C05476=1184.490,135.905,-53.759,-178.491,6.283,148.692
C05477=1184.495,135.656,-53.738,-178.495,6.282,148.692
C05478=1184.501,135.407,-53.718,-178.497,6.280,148.693
C05479=1184.505,135.158,-53.698,-178.499,6.279,148.693
C05480=1184.509,134.909,-53.678,-178.502,6.277,148.694
C05481=1184.515,134.659,-53.657,-178.505,6.275,148.694
C05482=1184.519,134.410,-53.637,-178.508,6.274,148.695
C05483=1184.524,134.161,-53.617,-178.510,6.273,148.695
C05484=1184.529,133.912,-53.597,-178.513,6.271,148.695
C05485=1184.533,133.663,-53.577,-178.515,6.270,148.696
C05486=1184.538,133.414,-53.557,-178.519,6.268,148.696
C05487=1184.544,133.165,-53.536,-178.521,6.267,148.697
C05488=1184.548,132.897,-53.515,-178.523,6.266,148.697
C05489=1184.554,132.628,-53.493,-178.527,6.264,148.698
C05490=1184.559,132.359,-53.472,-178.529,6.262,148.698
C05491=1184.564,132.091,-53.449,-178.532,6.261,148.699
C05492=1184.569,131.841,-53.430,-178.535,6.259,148.699
C05493=1184.573,131.592,-53.409,-178.538,6.257,148.700
C05494=1184.578,131.342,-53.390,-178.540,6.257,148.700
C05495=1184.582,131.094,-53.369,-178.543,6.255,148.700
C05496=1184.587,130.844,-53.350,-178.546,6.253,148.701
C05497=1184.592,130.596,-53.330,-178.549,6.252,148.701
C05498=1184.597,130.346,-53.310,-178.551,6.251,148.702
C05499=1184.602,130.097,-53.289,-178.553,6.249,148.702
C05500=1184.607,129.847,-53.269,-178.557,6.248,148.703
C05501=1184.612,129.599,-53.249,-178.559,6.247,148.703
C05502=1184.617,129.349,-53.230,-178.561,6.245,148.704
C05503=1184.621,129.101,-53.209,-178.565,6.243,148.704
C05504=1184.626,128.851,-53.190,-178.567,6.242,148.705
C05505=1184.631,128.601,-53.170,-178.569,6.241,148.705
C05506=1184.636,128.353,-53.150,-178.572,6.239,148.705
C05507=1184.640,128.104,-53.130,-178.575,6.238,148.706
C05508=1184.645,127.855,-53.110,-178.577,6.237,148.706
C05509=1184.650,127.605,-53.090,-178.580,6.235,148.707
C05510=1184.655,127.356,-53.071,-178.583,6.233,148.707
C05511=1184.659,127.107,-53.051,-178.585,6.233,148.708
C05512=1184.664,126.858,-53.031,-178.588,6.231,148.708
C05513=1184.669,126.608,-53.011,-178.591,6.229,148.709
C05514=1184.674,126.360,-52.991,-178.593,6.227,148.709
C05515=1184.679,126.110,-52.972,-178.596,6.227,148.710
C05516=1184.683,125.861,-52.952,-178.599,6.225,148.710
C05517=1184.688,125.612,-52.932,-178.601,6.223,148.710
C05518=1184.693,125.363,-52.912,-178.604,6.223,148.711
C05519=1184.697,125.114,-52.893,-178.607,6.221,148.711
C05520=1184.702,124.865,-52.873,-178.609,6.219,148.712
C05521=1184.707,124.616,-52.854,-178.612,6.218,148.712
C05522=1184.712,124.366,-52.834,-178.615,6.217,148.713
C05523=1184.716,124.117,-52.814,-178.617,6.215,148.713
C05524=1184.721,123.867,-52.795,-178.620,6.214,148.714
C05525=1184.726,123.619,-52.775,-178.623,6.213,148.714
C05526=1184.731,123.369,-52.755,-178.625,6.211,148.715
C05527=1184.736,123.120,-52.735,-178.628,6.210,148.715
C05528=1184.741,122.871,-52.716,-178.630,6.208,148.716
C05529=1184.745,122.622,-52.697,-178.633,6.207,148.716
C05530=1184.749,122.373,-52.677,-178.636,6.206,148.717
C05531=1184.755,122.124,-52.657,-178.638,6.204,148.717
C05532=1184.760,121.874,-52.638,-178.641,6.203,148.718
C05533=1184.764,121.625,-52.618,-178.644,6.202,148.718
C05534=1184.770,121.376,-52.599,-178.646,6.200,148.718
C05535=1184.774,121.127,-52.580,-178.650,6.199,148.719
C05536=1184.779,120.878,-52.560,-178.652,6.198,148.719
C05537=1184.784,120.628,-52.541,-178.654,6.196,148.720
C05538=1184.788,120.379,-52.520,-178.657,6.194,148.720
C05539=1184.793,120.130,-52.501,-178.660,6.194,148.721
C05540=1184.797,119.881,-52.482,-178.662,6.192,148.721
C05541=1184.802,119.631,-52.462,-178.665,6.190,148.722
C05542=1184.808,119.383,-52.443,-178.668,6.190,148.722
C05543=1184.812,119.133,-52.423,-178.670,6.188,148.723
C05544=1184.818,118.884,-52.404,-178.673,6.186,148.723
C05545=1184.822,118.635,-52.385,-178.676,6.186,148.724
C05546=1184.826,118.385,-52.365,-178.678,6.184,148.724
C05547=1184.832,118.136,-52.346,-178.680,6.183,148.725
C05548=1184.837,117.887,-52.327,-178.684,6.182,148.725
C05549=1184.841,117.638,-52.308,-178.686,6.180,148.726
C05550=1184.846,117.389,-52.288,-178.689,6.179,148.726
C05551=1184.851,117.140,-52.269,-178.692,6.178,148.727
C05552=1184.855,116.891,-52.250,-178.694,6.176,148.727
C05553=1184.860,116.640,-52.231,-178.697,6.175,148.727
C05554=1184.866,116.392,-52.212,-178.700,6.174,148.728
C05555=1184.870,116.142,-52.192,-178.702,6.172,148.728
C05556=1184.875,115.893,-52.173,-178.705,6.171,148.729
C05557=1184.880,115.644,-52.154,-178.708,6.170,148.729
C05558=1184.885,115.395,-52.134,-178.710,6.169,148.730
C05559=1184.889,115.146,-52.115,-178.713,6.167,148.730
C05560=1184.894,114.897,-52.096,-178.716,6.165,148.731
C05561=1184.899,114.647,-52.076,-178.718,6.165,148.731
C05562=1184.904,114.398,-52.058,-178.721,6.163,148.732
C05563=1184.909,114.149,-52.039,-178.723,6.162,148.732
C05564=1184.913,113.900,-52.020,-178.726,6.161,148.733
C05565=1184.918,113.650,-52.000,-178.729,6.159,148.733
C05566=1184.923,113.402,-51.981,-178.731,6.158,148.734
C05567=1184.928,113.152,-51.963,-178.734,6.156,148.734
C05568=1184.933,112.903,-51.943,-178.736,6.156,148.735
C05569=1184.937,112.654,-51.924,-178.739,6.154,148.735
C05570=1184.942,112.405,-51.905,-178.742,6.152,148.736
C05571=1184.948,112.155,-51.886,-178.744,6.151,148.736
C05572=1184.952,111.906,-51.867,-178.747,6.150,148.737
C05573=1184.957,111.656,-51.848,-178.749,6.149,148.737
C05574=1184.961,111.408,-51.829,-178.753,6.148,148.738
C05575=1184.967,111.158,-51.810,-178.755,6.146,148.738
C05576=1184.971,110.909,-51.791,-178.757,6.145,148.739
C05577=1184.976,110.660,-51.772,-178.761,6.144,148.739
C05578=1184.982,110.410,-51.753,-178.763,6.143,148.740
C05579=1184.986,110.162,-51.734,-178.765,6.141,148.740
C05580=1184.991,109.912,-51.715,-178.769,6.140,148.741
C05581=1184.996,109.663,-51.697,-178.771,6.139,148.741
C05582=1185.001,109.413,-51.677,-178.773,6.137,148.741
C05583=1185.005,109.165,-51.658,-178.776,6.136,148.742
C05584=1185.010,108.914,-51.640,-178.779,6.135,148.743
C05585=1185.015,108.666,-51.621,-178.782,6.133,148.743
C05586=1185.020,108.417,-51.603,-178.784,6.132,148.744
C05587=1185.024,108.167,-51.583,-178.787,6.131,148.744
C05588=1185.029,107.919,-51.564,-178.789,6.130,148.745
C05589=1185.034,107.668,-51.546,-178.792,6.128,148.745
C05590=1185.039,107.420,-51.527,-178.794,6.127,148.745
C05591=1185.044,107.170,-51.508,-178.797,6.126,148.746
C05592=1185.049,106.902,-51.488,-178.800,6.124,148.746
C05593=1185.054,106.633,-51.468,-178.803,6.124,148.747
C05594=1185.060,106.366,-51.447,-178.806,6.122,148.748
C05595=1185.064,106.097,-51.427,-178.809,6.121,148.748
C05596=1185.070,105.847,-51.409,-178.812,6.119,148.749
C05597=1185.075,105.599,-51.390,-178.814,6.118,148.749
C05598=1185.079,105.349,-51.372,-178.817,6.117,148.750
C05599=1185.084,105.100,-51.352,-178.819,6.116,148.750
C05600=1185.089,104.850,-51.334,-178.822,6.114,148.751
C05601=1185.093,104.601,-51.315,-178.824,6.113,148.751
C05602=1185.099,104.352,-51.297,-178.827,6.112,148.752
C05603=1185.103,104.103,-51.278,-178.830,6.111,148.752
C05604=1185.108,103.853,-51.260,-178.833,6.110,148.753
C05605=1185.113,103.604,-51.241,-178.835,6.109,148.753
C05606=1185.117,103.355,-51.222,-178.838,6.107,148.754
C05607=1185.122,103.106,-51.204,-178.841,6.106,148.754
C05608=1185.128,102.857,-51.185,-178.843,6.105,148.755
C05609=1185.133,102.607,-51.167,-178.846,6.103,148.755
C05610=1185.137,102.358,-51.148,-178.848,6.103,148.756
C05611=1185.142,102.109,-51.129,-178.851,6.101,148.756
C05612=1185.147,101.860,-51.111,-178.854,6.100,148.757
C05613=1185.151,101.610,-51.093,-178.856,6.099,148.757
C05614=1185.157,101.361,-51.074,-178.859,6.098,148.758
C05615=1185.162,101.112,-51.056,-178.862,6.096,148.758
C05616=1185.166,100.862,-51.037,-178.864,6.096,148.759
C05617=1185.171,100.613,-51.019,-178.867,6.094,148.759
C05618=1185.176,100.364,-51.000,-178.869,6.093,148.760
C05619=1185.181,100.115,-50.982,-178.872,6.092,148.760
C05620=1185.185,99.865,-50.964,-178.874,6.091,148.761
C05621=1185.190,99.616,-50.945,-178.878,6.089,148.761
C05622=1185.196,99.367,-50.926,-178.880,6.088,148.762
C05623=1185.201,99.117,-50.908,-178.883,6.087,148.762
C05624=1185.205,98.868,-50.890,-178.886,6.085,148.763
C05625=1185.210,98.619,-50.871,-178.888,6.084,148.763
C05626=1185.214,98.370,-50.853,-178.891,6.083,148.764
C05627=1185.220,98.120,-50.835,-178.893,6.082,148.764
C05628=1185.224,97.870,-50.816,-178.896,6.081,148.765
C05629=1185.229,97.621,-50.798,-178.898,6.080,148.765
C05630=1185.234,97.372,-50.781,-178.902,6.078,148.766
C05631=1185.239,97.124,-50.762,-178.904,6.078,148.766
C05632=1185.244,96.874,-50.744,-178.906,6.076,148.767
C05633=1185.249,96.624,-50.725,-178.909,6.075,148.767
C05634=1185.254,96.375,-50.707,-178.912,6.074,148.768
C05635=1185.259,96.126,-50.689,-178.914,6.073,148.769
C05636=1185.264,95.877,-50.671,-178.917,6.071,148.769
C05637=1185.268,95.628,-50.653,-178.920,6.071,148.770
C05638=1185.273,95.378,-50.635,-178.922,6.069,148.770
C05639=1185.278,95.128,-50.617,-178.925,6.068,148.770
C05640=1185.283,94.879,-50.598,-178.928,6.067,148.771
C05641=1185.288,94.630,-50.579,-178.930,6.066,148.771
C05642=1185.293,94.381,-50.561,-178.933,6.065,148.772
C05643=1185.298,94.132,-50.543,-178.935,6.063,148.773
C05644=1185.302,93.882,-50.525,-178.938,6.063,148.773
C05645=1185.307,93.633,-50.507,-178.941,6.061,148.774
C05646=1185.312,93.384,-50.489,-178.943,6.061,148.774
C05647=1185.317,93.135,-50.471,-178.946,6.059,148.775
C05648=1185.322,92.885,-50.453,-178.949,6.058,148.775
C05649=1185.327,92.636,-50.435,-178.951,6.057,148.776
C05650=1185.332,92.387,-50.417,-178.953,6.056,148.776
C05651=1185.336,92.137,-50.399,-178.957,6.054,148.777
C05652=1185.341,91.887,-50.382,-178.959,6.053,148.777
C05653=1185.346,91.638,-50.364,-178.962,6.052,148.778
C05654=1185.351,91.389,-50.346,-178.964,6.051,148.778
C05655=1185.356,91.140,-50.328,-178.967,6.050,148.779
C05656=1185.361,90.891,-50.310,-178.969,6.049,148.779
C05657=1185.366,90.642,-50.292,-178.973,6.048,148.780
C05658=1185.371,90.392,-50.274,-178.975,6.047,148.780
C05659=1185.375,90.143,-50.255,-178.977,6.046,148.781
C05660=1185.380,89.893,-50.237,-178.980,6.044,148.781
C05661=1185.385,89.644,-50.219,-178.983,6.044,148.782
C05662=1185.390,89.394,-50.202,-178.985,6.042,148.783
C05663=1185.395,89.145,-50.184,-178.988,6.041,148.783
C05664=1185.400,88.896,-50.166,-178.991,6.040,148.784
C05665=1185.405,88.647,-50.148,-178.993,6.039,148.784
C05666=1185.410,88.398,-50.130,-178.996,6.038,148.785
C05667=1185.414,88.148,-50.112,-178.998,6.037,148.785
C05668=1185.420,87.899,-50.095,-179.001,6.035,148.786
C05669=1185.425,87.650,-50.077,-179.004,6.034,148.786
C05670=1185.430,87.400,-50.059,-179.006,6.034,148.787
C05671=1185.434,87.151,-50.042,-179.009,6.032,148.787
C05672=1185.439,86.902,-50.024,-179.012,6.032,148.788
C05673=1185.444,86.653,-50.006,-179.014,6.030,148.788
C05674=1185.449,86.403,-49.988,-179.017,6.029,148.789
C05675=1185.454,86.154,-49.970,-179.020,6.028,148.789
C05676=1185.459,85.904,-49.953,-179.022,6.027,148.790
C05677=1185.464,85.655,-49.935,-179.024,6.026,148.790
C05678=1185.469,85.406,-49.917,-179.028,6.025,148.791
C05679=1185.473,85.157,-49.901,-179.030,6.024,148.792
C05680=1185.478,84.907,-49.883,-179.033,6.022,148.792
C05681=1185.483,84.658,-49.865,-179.035,6.022,148.793
C05682=1185.488,84.408,-49.847,-179.038,6.020,148.793
C05683=1185.493,84.159,-49.829,-179.040,6.019,148.794
C05684=1185.498,83.910,-49.811,-179.043,6.019,148.794
C05685=1185.503,83.661,-49.795,-179.046,6.017,148.795
C05686=1185.507,83.411,-49.777,-179.048,6.016,148.795
C05687=1185.512,83.162,-49.759,-179.051,6.015,148.796
C05688=1185.518,82.912,-49.741,-179.054,6.014,148.796
C05689=1185.522,82.664,-49.724,-179.056,6.013,148.797
C05690=1185.527,82.414,-49.707,-179.059,6.012,148.798
C05691=1185.532,82.165,-49.689,-179.061,6.011,148.798
C05692=1185.537,81.915,-49.672,-179.064,6.010,148.799
C05693=1185.542,81.666,-49.654,-179.067,6.009,148.799
C05694=1185.546,81.417,-49.636,-179.070,6.007,148.800
C05695=1185.551,81.167,-49.619,-179.072,6.007,148.800
C05696=1185.556,80.899,-49.600,-179.075,6.005,148.801
C05697=1185.562,80.630,-49.581,-179.078,6.005,148.801
C05698=1185.567,80.362,-49.563,-179.080,6.003,148.802
C05699=1185.572,80.094,-49.544,-179.083,6.002,148.803
C05700=1185.577,79.844,-49.526,-179.086,6.001,148.803
C05701=1185.582,79.595,-49.508,-179.088,6.000,148.804
C05702=1185.587,79.345,-49.492,-179.091,6.000,148.804
C05703=1185.592,79.096,-49.474,-179.094,5.998,148.805
C05704=1185.597,78.846,-49.457,-179.096,5.997,148.805
C05705=1185.602,78.597,-49.440,-179.099,5.996,148.806
C05706=1185.607,78.348,-49.422,-179.102,5.995,148.806
C05707=1185.612,78.099,-49.405,-179.104,5.994,148.807
C05708=1185.616,77.850,-49.388,-179.107,5.993,148.807
C05709=1185.622,77.600,-49.370,-179.109,5.992,148.808
C05710=1185.627,77.350,-49.353,-179.112,5.991,148.809
C05711=1185.631,77.101,-49.336,-179.115,5.990,148.809
C05712=1185.636,76.851,-49.318,-179.117,5.989,148.810
C05713=1185.642,76.603,-49.301,-179.120,5.987,148.810
C05714=1185.646,76.353,-49.284,-179.123,5.987,148.811
C05715=1185.651,76.104,-49.267,-179.125,5.986,148.811
C05716=1185.656,75.855,-49.249,-179.128,5.985,148.812
C05717=1185.661,75.605,-49.232,-179.130,5.984,148.812
C05718=1185.666,75.355,-49.215,-179.133,5.983,148.813
C05719=1185.670,75.106,-49.198,-179.136,5.982,148.814
C05720=1185.676,74.857,-49.181,-179.138,5.981,148.814
C05721=1185.680,74.608,-49.164,-179.141,5.980,148.815
C05722=1185.686,74.358,-49.147,-179.143,5.979,148.815
C05723=1185.690,74.109,-49.129,-179.146,5.978,148.816
C05724=1185.695,73.859,-49.112,-179.149,5.976,148.816
C05725=1185.700,73.610,-49.095,-179.151,5.976,148.817
C05726=1185.705,73.361,-49.079,-179.153,5.975,148.817
C05727=1185.710,73.112,-49.061,-179.157,5.974,148.818
C05728=1185.715,72.862,-49.044,-179.159,5.973,148.818
C05729=1185.720,72.612,-49.027,-179.161,5.972,148.819
C05730=1185.725,72.363,-49.010,-179.164,5.970,148.819
C05731=1185.730,72.114,-48.992,-179.167,5.970,148.820
C05732=1185.734,71.865,-48.976,-179.169,5.969,148.821
C05733=1185.740,71.615,-48.958,-179.172,5.968,148.821
C05734=1185.744,71.366,-48.942,-179.175,5.967,148.822
C05735=1185.750,71.116,-48.925,-179.177,5.966,148.822
C05736=1185.754,70.867,-48.908,-179.180,5.965,148.823
C05737=1185.759,70.618,-48.891,-179.182,5.964,148.823
C05738=1185.764,70.368,-48.874,-179.185,5.963,148.824
C05739=1185.769,70.120,-48.857,-179.188,5.962,148.824
C05740=1185.774,69.870,-48.840,-179.190,5.961,148.825
C05741=1185.779,69.620,-48.823,-179.193,5.961,148.826
C05742=1185.784,69.370,-48.806,-179.196,5.959,148.826
C05743=1185.789,69.122,-48.790,-179.198,5.958,148.827
C05744=1185.794,68.872,-48.772,-179.200,5.958,148.827
C05745=1185.799,68.622,-48.756,-179.204,5.956,148.828
C05746=1185.803,68.373,-48.739,-179.206,5.955,148.828
C05747=1185.809,68.124,-48.722,-179.208,5.955,148.829
C05748=1185.813,67.874,-48.706,-179.211,5.953,148.829
C05749=1185.819,67.625,-48.688,-179.214,5.953,148.830
C05750=1185.824,67.376,-48.672,-179.216,5.952,148.831
C05751=1185.828,67.126,-48.655,-179.219,5.950,148.831
C05752=1185.833,66.876,-48.638,-179.222,5.950,148.832
C05753=1185.838,66.627,-48.621,-179.224,5.949,148.832
C05754=1185.843,66.378,-48.605,-179.227,5.948,148.833
C05755=1185.848,66.128,-48.588,-179.229,5.947,148.833
C05756=1185.853,65.879,-48.571,-179.232,5.946,148.834
C05757=1185.858,65.630,-48.555,-179.235,5.945,148.835
C05758=1185.863,65.380,-48.538,-179.237,5.944,148.835
C05759=1185.867,65.131,-48.521,-179.240,5.943,148.836
C05760=1185.872,64.882,-48.505,-179.242,5.942,148.836
C05761=1185.878,64.632,-48.487,-179.245,5.941,148.837
C05762=1185.882,64.383,-48.471,-179.247,5.940,148.837
C05763=1185.887,64.134,-48.454,-179.250,5.940,148.838
C05764=1185.892,63.885,-48.438,-179.253,5.938,148.839
C05765=1185.897,63.635,-48.420,-179.255,5.937,148.839
C05766=1185.902,63.386,-48.404,-179.258,5.937,148.840
C05767=1185.907,63.136,-48.388,-179.261,5.935,148.840
C05768=1185.912,62.886,-48.371,-179.263,5.935,148.841
C05769=1185.917,62.637,-48.355,-179.266,5.934,148.842
C05770=1185.922,62.388,-48.338,-179.268,5.933,148.842
C05771=1185.927,62.139,-48.322,-179.271,5.932,148.843
C05772=1185.932,61.889,-48.304,-179.273,5.931,148.843
C05773=1185.937,61.639,-48.288,-179.276,5.931,148.844
C05774=1185.942,61.390,-48.272,-179.279,5.929,148.844
C05775=1185.946,61.141,-48.255,-179.281,5.928,148.845
C05776=1185.951,60.892,-48.239,-179.284,5.928,148.845
C05777=1185.957,60.642,-48.223,-179.286,5.927,148.846
C05778=1185.961,60.392,-48.206,-179.289,5.926,148.847
C05779=1185.966,60.143,-48.190,-179.292,5.925,148.847
C05780=1185.971,59.894,-48.173,-179.294,5.924,148.848
C05781=1185.976,59.644,-48.157,-179.297,5.923,148.848
C05782=1185.982,59.395,-48.140,-179.300,5.922,148.849
C05783=1185.987,59.146,-48.124,-179.302,5.921,148.849
C05784=1185.991,58.896,-48.107,-179.304,5.920,148.850
C05785=1185.996,58.646,-48.091,-179.308,5.919,148.851
C05786=1186.001,58.398,-48.075,-179.310,5.919,148.851
C05787=1186.005,58.148,-48.058,-179.312,5.918,148.852
C05788=1186.012,57.898,-48.042,-179.315,5.917,148.852
C05789=1186.016,57.649,-48.025,-179.318,5.915,148.853
C05790=1186.021,57.400,-48.009,-179.320,5.915,148.853
C05791=1186.026,57.150,-47.993,-179.323,5.914,148.854
C05792=1186.031,56.901,-47.977,-179.325,5.914,148.855
C05793=1186.035,56.652,-47.960,-179.328,5.912,148.855
C05794=1186.041,56.402,-47.945,-179.331,5.911,148.856
C05795=1186.045,56.153,-47.928,-179.333,5.911,148.856
C05796=1186.051,55.903,-47.912,-179.336,5.910,148.857
C05797=1186.056,55.654,-47.895,-179.339,5.909,148.857
C05798=1186.061,55.405,-47.879,-179.341,5.908,148.858
C05799=1186.066,55.155,-47.863,-179.344,5.908,148.859
C05800=1186.071,54.886,-47.846,-179.347,5.906,148.859
C05801=1186.076,54.618,-47.828,-179.349,5.905,148.860
C05802=1186.082,54.349,-47.811,-179.352,5.905,148.860
C05803=1186.087,54.081,-47.794,-179.355,5.903,148.861
C05804=1186.092,53.831,-47.777,-179.357,5.903,148.862
C05805=1186.097,53.582,-47.761,-179.360,5.902,148.862
C05806=1186.101,53.332,-47.745,-179.363,5.901,148.863
C05807=1186.107,53.083,-47.729,-179.365,5.900,148.863
C05808=1186.111,52.833,-47.712,-179.368,5.899,148.864
C05809=1186.117,52.584,-47.697,-179.370,5.898,148.864
C05810=1186.122,52.335,-47.681,-179.373,5.898,148.865
C05811=1186.127,52.085,-47.665,-179.376,5.897,148.866
C05812=1186.132,51.836,-47.648,-179.378,5.896,148.866
C05813=1186.136,51.586,-47.632,-179.381,5.895,148.867
C05814=1186.142,51.338,-47.616,-179.383,5.895,148.868
C05815=1186.146,51.087,-47.600,-179.386,5.893,148.868
C05816=1186.152,50.838,-47.584,-179.389,5.892,148.869
C05817=1186.156,50.589,-47.568,-179.391,5.892,148.869
C05818=1186.162,50.339,-47.552,-179.393,5.891,148.870
C05819=1186.167,50.090,-47.536,-179.396,5.891,148.870
C05820=1186.171,49.840,-47.520,-179.399,5.889,148.871
C05821=1186.177,49.591,-47.504,-179.401,5.888,148.872
C05822=1186.181,49.341,-47.488,-179.404,5.888,148.872
C05823=1186.187,49.092,-47.472,-179.406,5.887,148.873
C05824=1186.192,48.843,-47.457,-179.409,5.886,148.873
C05825=1186.196,48.593,-47.440,-179.412,5.885,148.874
C05826=1186.201,48.344,-47.425,-179.414,5.884,148.874
C05827=1186.206,48.094,-47.409,-179.417,5.884,148.875
C05828=1186.211,47.845,-47.393,-179.419,5.883,148.876
C05829=1186.216,47.596,-47.377,-179.422,5.881,148.876
C05830=1186.221,47.346,-47.361,-179.425,5.881,148.877
C05831=1186.226,47.097,-47.345,-179.427,5.880,148.877
C05832=1186.231,46.847,-47.329,-179.430,5.880,148.878
C05833=1186.236,46.598,-47.314,-179.432,5.879,148.879
C05834=1186.241,46.348,-47.298,-179.435,5.877,148.879
C05835=1186.246,46.099,-47.282,-179.438,5.877,148.880
C05836=1186.251,45.849,-47.266,-179.440,5.876,148.880
C05837=1186.256,45.600,-47.250,-179.443,5.875,148.881
C05838=1186.261,45.350,-47.234,-179.445,5.875,148.882
C05839=1186.266,45.101,-47.219,-179.447,5.874,148.882
C05840=1186.271,44.852,-47.203,-179.451,5.873,148.883
C05841=1186.276,44.602,-47.187,-179.453,5.872,148.883
C05842=1186.281,44.352,-47.172,-179.455,5.871,148.884
C05843=1186.286,44.103,-47.156,-179.458,5.871,148.884
C05844=1186.291,43.853,-47.141,-179.461,5.870,148.885
C05845=1186.296,43.604,-47.124,-179.463,5.869,148.886
C05846=1186.301,43.355,-47.109,-179.466,5.868,148.886
C05847=1186.306,43.105,-47.093,-179.469,5.868,148.887
C05848=1186.311,42.856,-47.077,-179.471,5.867,148.887
C05849=1186.316,42.606,-47.062,-179.473,5.866,148.888
C05850=1186.321,42.357,-47.047,-179.476,5.866,148.889
C05851=1186.326,42.107,-47.031,-179.479,5.864,148.889
C05852=1186.331,41.858,-47.015,-179.481,5.863,148.890
C05853=1186.336,41.609,-46.999,-179.484,5.863,148.891
C05854=1186.341,41.359,-46.983,-179.486,5.862,148.891
C05855=1186.346,41.110,-46.968,-179.489,5.862,148.892
C05856=1186.351,40.860,-46.953,-179.492,5.861,148.892
C05857=1186.356,40.611,-46.937,-179.494,5.859,148.893
C05858=1186.361,40.361,-46.921,-179.497,5.859,148.893
C05859=1186.366,40.112,-46.906,-179.499,5.858,148.894
C05860=1186.371,39.862,-46.891,-179.502,5.857,148.895
C05861=1186.376,39.613,-46.875,-179.504,5.857,148.895
C05862=1186.381,39.363,-46.859,-179.506,5.856,148.896
C05863=1186.386,39.114,-46.844,-179.510,5.855,148.896
C05864=1186.391,38.864,-46.829,-179.512,5.854,148.897
C05865=1186.396,38.615,-46.813,-179.515,5.853,148.897
C05866=1186.400,38.365,-46.798,-179.517,5.853,148.898
C05867=1186.406,38.116,-46.782,-179.520,5.852,148.899
C05868=1186.411,37.866,-46.766,-179.522,5.851,148.899
C05869=1186.416,37.617,-46.751,-179.525,5.851,148.900
C05870=1186.421,37.368,-46.736,-179.528,5.850,148.901
C05871=1186.425,37.118,-46.721,-179.530,5.849,148.901
C05872=1186.431,36.868,-46.706,-179.533,5.848,148.902
C05873=1186.436,36.619,-46.690,-179.535,5.848,148.902
C05874=1186.441,36.370,-46.675,-179.537,5.847,148.903
C05875=1186.446,36.120,-46.659,-179.540,5.846,148.904
C05876=1186.450,35.870,-46.644,-179.543,5.846,148.904
C05877=1186.456,35.621,-46.629,-179.545,5.844,148.905
C05878=1186.461,35.372,-46.613,-179.548,5.844,148.905
C05879=1186.466,35.123,-46.598,-179.551,5.843,148.906
C05880=1186.472,34.873,-46.583,-179.553,5.842,148.906
C05881=1186.476,34.623,-46.568,-179.556,5.842,148.907
C05882=1186.481,34.373,-46.552,-179.558,5.841,148.908
C05883=1186.486,34.124,-46.537,-179.560,5.840,148.908
C05884=1186.491,33.875,-46.522,-179.563,5.840,148.909
C05885=1186.496,33.625,-46.506,-179.566,5.839,148.910
C05886=1186.501,33.376,-46.492,-179.569,5.838,148.910
C05887=1186.507,33.126,-46.476,-179.571,5.837,148.911
C05888=1186.511,32.877,-46.461,-179.574,5.837,148.911
C05889=1186.516,32.627,-46.445,-179.576,5.836,148.912
C05890=1186.521,32.377,-46.431,-179.578,5.835,148.912
C05891=1186.527,32.128,-46.415,-179.581,5.835,148.913
C05892=1186.531,31.879,-46.400,-179.584,5.834,148.914
C05893=1186.537,31.630,-46.385,-179.586,5.833,148.914
C05894=1186.541,31.380,-46.370,-179.589,5.832,148.915
C05895=1186.547,31.130,-46.355,-179.592,5.832,148.916
C05896=1186.552,30.881,-46.340,-179.594,5.831,148.916
C05897=1186.556,30.632,-46.325,-179.597,5.830,148.917
C05898=1186.561,30.382,-46.310,-179.599,5.830,148.917
C05899=1186.566,30.132,-46.295,-179.601,5.829,148.918
C05900=1186.571,29.883,-46.279,-179.604,5.828,148.919
C05901=1186.576,29.633,-46.265,-179.607,5.828,148.919
C05902=1186.582,29.384,-46.249,-179.609,5.827,148.920
C05903=1186.586,29.135,-46.234,-179.612,5.826,148.920
C05904=1186.592,28.866,-46.218,-179.615,5.825,148.921
C05905=1186.597,28.597,-46.202,-179.617,5.825,148.922
C05906=1186.603,28.328,-46.186,-179.620,5.824,148.922
C05907=1186.608,28.059,-46.170,-179.623,5.823,148.923
C05908=1186.613,27.810,-46.155,-179.625,5.822,148.924
C05909=1186.618,27.561,-46.140,-179.628,5.822,148.924
C05910=1186.623,27.311,-46.125,-179.631,5.821,148.925
C05911=1186.629,27.061,-46.110,-179.633,5.820,148.925
C05912=1186.634,26.812,-46.095,-179.635,5.820,148.926
C05913=1186.638,26.563,-46.080,-179.638,5.819,148.927
C05914=1186.644,26.313,-46.065,-179.641,5.819,148.927
C05915=1186.649,26.064,-46.051,-179.643,5.818,148.928
C05916=1186.653,25.814,-46.036,-179.646,5.817,148.929
C05917=1186.658,25.564,-46.020,-179.648,5.817,148.929
C05918=1186.663,25.315,-46.005,-179.651,5.815,148.930
C05919=1186.668,25.065,-45.991,-179.654,5.815,148.930
C05920=1186.673,24.816,-45.976,-179.656,5.814,148.931
C05921=1186.678,24.566,-45.961,-179.658,5.813,148.931
C05922=1186.683,24.317,-45.946,-179.661,5.813,148.932
C05923=1186.689,24.067,-45.931,-179.664,5.812,148.933
C05924=1186.693,23.818,-45.916,-179.666,5.811,148.933
C05925=1186.698,23.568,-45.902,-179.669,5.811,148.934
C05926=1186.703,23.318,-45.888,-179.671,5.810,148.935
C05927=1186.709,23.069,-45.872,-179.674,5.810,148.935
C05928=1186.714,22.819,-45.858,-179.676,5.809,148.936
C05929=1186.718,22.570,-45.843,-179.679,5.809,148.936
C05930=1186.724,22.321,-45.828,-179.681,5.808,148.937
C05931=1186.729,22.072,-45.813,-179.683,5.807,148.938
C05932=1186.734,21.822,-45.799,-179.686,5.807,148.938
C05933=1186.739,21.572,-45.785,-179.689,5.805,148.939
C05934=1186.744,21.323,-45.769,-179.692,5.805,148.940
C05935=1186.749,21.073,-45.755,-179.694,5.804,148.940
C05936=1186.754,20.824,-45.740,-179.697,5.804,148.941
C05937=1186.759,20.574,-45.726,-179.699,5.803,148.941
C05938=1186.764,20.325,-45.711,-179.702,5.802,148.942
C05939=1186.769,20.075,-45.696,-179.704,5.802,148.943
C05940=1186.774,19.825,-45.682,-179.707,5.801,148.943
C05941=1186.779,19.576,-45.667,-179.709,5.800,148.944
C05942=1186.784,19.327,-45.652,-179.712,5.800,148.944
C05943=1186.789,19.077,-45.638,-179.714,5.799,148.945
C05944=1186.795,18.827,-45.623,-179.717,5.799,148.946
C05945=1186.799,18.577,-45.609,-179.719,5.798,148.946
C05946=1186.805,18.329,-45.594,-179.722,5.798,148.947
C05947=1186.810,18.079,-45.580,-179.724,5.797,148.948
C05948=1186.815,17.829,-45.566,-179.727,5.796,148.948
C05949=1186.820,17.580,-45.551,-179.729,5.796,148.949
C05950=1186.825,17.330,-45.536,-179.732,5.795,148.949
C05951=1186.830,17.081,-45.522,-179.735,5.795,148.950
C05952=1186.835,16.831,-45.507,-179.737,5.794,148.951
C05953=1186.840,16.581,-45.493,-179.739,5.793,148.951
C05954=1186.844,16.332,-45.478,-179.742,5.793,148.952
C05955=1186.849,16.082,-45.464,-179.744,5.792,148.952
C05956=1186.855,15.833,-45.450,-179.747,5.792,148.953
C05957=1186.860,15.584,-45.436,-179.750,5.790,148.954
C05958=1186.865,15.334,-45.421,-179.753,5.790,148.954
C05959=1186.870,15.084,-45.406,-179.755,5.789,148.955
C05960=1186.875,14.835,-45.391,-179.758,5.788,148.956
C05961=1186.880,14.585,-45.377,-179.760,5.788,148.956
C05962=1186.885,14.335,-45.363,-179.762,5.787,148.957
C05963=1186.891,14.086,-45.349,-179.765,5.787,148.957
C05964=1186.896,13.837,-45.335,-179.768,5.786,148.958
C05965=1186.901,13.587,-45.320,-179.770,5.786,148.959
C05966=1186.905,13.338,-45.305,-179.772,5.785,148.959
C05967=1186.910,13.088,-45.291,-179.775,5.784,148.960
C05968=1186.915,12.838,-45.277,-179.778,5.784,148.961
C05969=1186.921,12.589,-45.263,-179.780,5.783,148.961
C05970=1186.926,12.340,-45.249,-179.783,5.782,148.962
C05971=1186.931,12.090,-45.234,-179.785,5.782,148.962
C05972=1186.936,11.840,-45.220,-179.788,5.781,148.963
C05973=1186.941,11.591,-45.206,-179.790,5.781,148.964
C05974=1186.946,11.342,-45.192,-179.793,5.780,148.964
C05975=1186.951,11.092,-45.178,-179.795,5.780,148.965
C05976=1186.956,10.842,-45.163,-179.798,5.779,148.966
C05977=1186.961,10.592,-45.149,-179.800,5.778,148.966
C05978=1186.966,10.343,-45.135,-179.803,5.778,148.967
C05979=1186.971,10.094,-45.121,-179.805,5.777,148.967
C05980=1186.976,9.844,-45.107,-179.808,5.776,148.968
C05981=1186.981,9.594,-45.092,-179.810,5.776,148.969
C05982=1186.986,9.345,-45.078,-179.813,5.775,148.969
C05983=1186.992,9.096,-45.064,-179.816,5.775,148.970
C05984=1186.997,8.846,-45.050,-179.818,5.774,148.970
C05985=1187.002,8.596,-45.036,-179.820,5.774,148.971
C05986=1187.007,8.346,-45.021,-179.823,5.773,148.972
C05987=1187.012,8.097,-45.007,-179.825,5.772,148.972
C05988=1187.017,7.848,-44.993,-179.828,5.772,148.973
C05989=1187.022,7.598,-44.979,-179.830,5.771,148.974
C05990=1187.026,7.349,-44.965,-179.833,5.771,148.974
C05991=1187.032,7.100,-44.951,-179.835,5.770,148.975
C05992=1187.037,6.850,-44.937,-179.838,5.769,148.975
C05993=1187.042,6.600,-44.923,-179.841,5.769,148.976
C05994=1187.047,6.350,-44.909,-179.843,5.768,148.977
C05995=1187.053,6.101,-44.895,-179.845,5.768,148.977
C05996=1187.058,5.851,-44.881,-179.848,5.767,148.978
C05997=1187.063,5.601,-44.867,-179.850,5.767,148.979
C05998=1187.067,5.353,-44.853,-179.852,5.767,148.979
C05999=1187.072,5.103,-44.839,-179.855,5.766,148.980
C06000=1187.078,4.853,-44.826,-179.858,5.766,148.980
C06001=1187.083,4.603,-44.811,-179.860,5.765,148.981
C06002=1187.088,4.354,-44.797,-179.862,5.764,148.982
C06003=1187.093,4.104,-44.783,-179.865,5.764,148.982
C06004=1187.097,3.855,-44.769,-179.868,5.763,148.983
C06005=1187.103,3.605,-44.756,-179.870,5.763,148.984
C06006=1187.108,3.355,-44.742,-179.873,5.762,148.984
C06007=1187.113,3.106,-44.728,-179.875,5.762,148.985
C06008=1187.119,2.837,-44.713,-179.878,5.761,148.985
C06009=1187.125,2.568,-44.698,-179.881,5.761,148.986
C06010=1187.130,2.298,-44.683,-179.884,5.759,148.987
C06011=1187.135,2.029,-44.668,-179.886,5.759,148.988
C06012=1187.140,1.780,-44.655,-179.889,5.758,148.988
C06013=1187.145,1.530,-44.640,-179.891,5.758,148.989
C06014=1187.150,1.281,-44.626,-179.893,5.758,148.989
C06015=1187.156,1.031,-44.613,-179.896,5.757,148.990
C06016=1187.161,0.781,-44.599,-179.899,5.757,148.991
C06017=1187.165,0.532,-44.585,-179.901,5.756,148.991
C06018=1187.171,0.282,-44.572,-179.903,5.756,148.992
C06019=1187.176,0.033,-44.558,-179.906,5.755,148.993
C06020=1187.181,-0.216,-44.544,-179.909,5.755,148.993
C06021=1187.186,-0.466,-44.531,-179.911,5.754,148.994
C06022=1187.191,-0.716,-44.516,-179.914,5.753,148.994
C06023=1187.197,-0.965,-44.503,-179.916,5.753,148.995
C06024=1187.201,-1.215,-44.490,-179.918,5.752,148.996
C06025=1187.206,-1.465,-44.475,-179.921,5.751,148.996
C06026=1187.212,-1.714,-44.462,-179.924,5.751,148.997
C06027=1187.216,-1.964,-44.448,-179.926,5.751,148.998
C06028=1187.222,-2.213,-44.434,-179.929,5.750,148.998
C06029=1187.227,-2.463,-44.421,-179.931,5.749,148.999
C06030=1187.232,-2.712,-44.408,-179.934,5.749,148.999
C06031=1187.237,-2.962,-44.394,-179.936,5.749,149.000
C06032=1187.242,-3.212,-44.380,-179.938,5.748,149.001
C06033=1187.247,-3.461,-44.366,-179.941,5.748,149.001
C06034=1187.252,-3.711,-44.353,-179.943,5.747,149.002
C06035=1187.258,-3.960,-44.339,-179.946,5.747,149.003
C06036=1187.262,-4.210,-44.326,-179.948,5.746,149.003
C06037=1187.268,-4.459,-44.312,-179.951,5.745,149.004
C06038=1187.273,-4.709,-44.299,-179.954,5.745,149.005
C06039=1187.277,-4.959,-44.285,-179.956,5.745,149.005
C06040=1187.283,-5.208,-44.272,-179.958,5.744,149.006
C06041=1187.288,-5.458,-44.257,-179.961,5.743,149.006
C06042=1187.293,-5.707,-44.245,-179.964,5.743,149.007
C06043=1187.298,-5.957,-44.230,-179.966,5.742,149.008
C06044=1187.303,-6.206,-44.218,-179.968,5.742,149.008
C06045=1187.308,-6.456,-44.204,-179.971,5.742,149.009
C06046=1187.314,-6.706,-44.190,-179.973,5.741,149.010
C06047=1187.319,-6.956,-44.177,-179.976,5.741,149.010
C06048=1187.324,-7.205,-44.164,-179.978,5.740,149.011
C06049=1187.329,-7.455,-44.151,-179.981,5.739,149.011
C06050=1187.334,-7.704,-44.137,-179.983,5.739,149.012
C06051=1187.339,-7.954,-44.124,-179.986,5.738,149.013
C06052=1187.344,-8.203,-44.110,-179.988,5.738,149.013
C06053=1187.349,-8.453,-44.097,-179.991,5.737,149.014
C06054=1187.355,-8.703,-44.084,-179.993,5.737,149.015
C06055=1187.359,-8.952,-44.070,-179.995,5.737,149.015
C06056=1187.365,-9.202,-44.057,-179.998,5.736,149.016
C06057=1187.369,-9.451,-44.043,180.000,5.736,149.017
C06058=1187.375,-9.701,-44.030,179.997,5.735,149.017
C06059=1187.380,-9.951,-44.016,179.995,5.734,149.018
C06060=1187.385,-10.200,-44.003,179.992,5.734,149.018
C06061=1187.390,-10.450,-43.989,179.989,5.734,149.019
C06062=1187.395,-10.699,-43.977,179.987,5.733,149.020
C06063=1187.400,-10.949,-43.963,179.985,5.732,149.020
C06064=1187.405,-11.198,-43.950,179.982,5.732,149.021
C06065=1187.410,-11.448,-43.937,179.980,5.732,149.022
C06066=1187.416,-11.698,-43.924,179.977,5.732,149.022
C06067=1187.421,-11.947,-43.910,179.975,5.731,149.023
C06068=1187.426,-12.197,-43.897,179.972,5.730,149.023
C06069=1187.431,-12.446,-43.884,179.970,5.730,149.024
C06070=1187.436,-12.696,-43.870,179.967,5.729,149.025
C06071=1187.441,-12.945,-43.857,179.965,5.729,149.025
C06072=1187.446,-13.196,-43.844,179.962,5.728,149.026
C06073=1187.451,-13.445,-43.831,179.960,5.728,149.027
C06074=1187.456,-13.694,-43.818,179.958,5.728,149.027
C06075=1187.462,-13.944,-43.804,179.955,5.727,149.028
C06076=1187.467,-14.193,-43.792,179.953,5.727,149.029
C06077=1187.472,-14.444,-43.778,179.950,5.726,149.029
C06078=1187.477,-14.693,-43.766,179.947,5.726,149.030
C06079=1187.481,-14.942,-43.752,179.945,5.725,149.030
C06080=1187.487,-15.192,-43.739,179.943,5.724,149.031
C06081=1187.492,-15.441,-43.726,179.940,5.724,149.032
C06082=1187.497,-15.692,-43.713,179.938,5.724,149.032
C06083=1187.503,-15.941,-43.700,179.936,5.723,149.033
C06084=1187.508,-16.190,-43.687,179.933,5.723,149.034
C06085=1187.513,-16.440,-43.673,179.930,5.722,149.034
C06086=1187.518,-16.689,-43.661,179.928,5.722,149.035
C06087=1187.522,-16.939,-43.648,179.926,5.721,149.035
C06088=1187.528,-17.189,-43.634,179.923,5.721,149.036
C06089=1187.533,-17.438,-43.622,179.921,5.721,149.037
C06090=1187.538,-17.688,-43.609,179.918,5.721,149.038
C06091=1187.544,-17.938,-43.596,179.916,5.720,149.038
C06092=1187.549,-18.187,-43.583,179.913,5.719,149.039
C06093=1187.553,-18.437,-43.570,179.911,5.719,149.039
C06094=1187.559,-18.687,-43.557,179.908,5.718,149.040
C06095=1187.564,-18.936,-43.544,179.906,5.718,149.041
C06096=1187.569,-19.186,-43.531,179.904,5.718,149.041
C06097=1187.574,-19.435,-43.517,179.901,5.717,149.042
C06098=1187.580,-19.685,-43.505,179.898,5.717,149.043
C06099=1187.584,-19.935,-43.492,179.896,5.716,149.043
C06100=1187.590,-20.184,-43.479,179.894,5.716,149.044
C06101=1187.595,-20.433,-43.466,179.891,5.715,149.045
C06102=1187.600,-20.684,-43.453,179.888,5.715,149.045
C06103=1187.605,-20.933,-43.440,179.887,5.715,149.046
C06104=1187.611,-21.182,-43.427,179.884,5.714,149.046
C06105=1187.615,-21.432,-43.414,179.881,5.714,149.047
C06106=1187.620,-21.682,-43.402,179.879,5.713,149.048
C06107=1187.625,-21.931,-43.389,179.877,5.712,149.048
C06108=1187.631,-22.181,-43.376,179.874,5.712,149.049
C06109=1187.636,-22.431,-43.363,179.872,5.712,149.050
C06110=1187.641,-22.680,-43.350,179.869,5.712,149.050
C06111=1187.646,-22.930,-43.338,179.867,5.711,149.051
C06112=1187.652,-23.200,-43.324,179.864,5.711,149.051
C06113=1187.657,-23.470,-43.310,179.862,5.710,149.052
C06114=1187.663,-23.739,-43.297,179.859,5.710,149.053
C06115=1187.668,-24.009,-43.283,179.856,5.709,149.054
C06116=1187.673,-24.258,-43.270,179.854,5.709,149.054
C06117=1187.679,-24.507,-43.258,179.851,5.708,149.055
C06118=1187.684,-24.758,-43.244,179.848,5.708,149.056
C06119=1187.689,-25.007,-43.231,179.847,5.708,149.056
C06120=1187.694,-25.256,-43.219,179.844,5.707,149.057
C06121=1187.699,-25.506,-43.206,179.841,5.707,149.058
C06122=1187.704,-25.756,-43.194,179.839,5.706,149.058
C06123=1187.709,-26.006,-43.181,179.837,5.706,149.059
C06124=1187.715,-26.255,-43.168,179.834,5.705,149.059
C06125=1187.720,-26.505,-43.156,179.832,5.706,149.060
C06126=1187.725,-26.755,-43.143,179.829,5.705,149.061
C06127=1187.730,-27.004,-43.130,179.827,5.704,149.061
C06128=1187.735,-27.254,-43.118,179.824,5.704,149.062
C06129=1187.740,-27.503,-43.106,179.822,5.703,149.063
C06130=1187.745,-27.753,-43.093,179.820,5.704,149.063
C06131=1187.750,-28.003,-43.080,179.817,5.703,149.064
C06132=1187.755,-28.253,-43.068,179.815,5.702,149.065
C06133=1187.761,-28.502,-43.055,179.812,5.702,149.065
C06134=1187.766,-28.751,-43.042,179.809,5.701,149.066
C06135=1187.771,-29.001,-43.029,179.807,5.701,149.066
C06136=1187.776,-29.251,-43.017,179.805,5.701,149.067
C06137=1187.782,-29.501,-43.005,179.803,5.701,149.068
C06138=1187.787,-29.750,-42.992,179.800,5.700,149.068
C06139=1187.792,-29.999,-42.980,179.798,5.699,149.069
C06140=1187.797,-30.249,-42.968,179.795,5.699,149.070
C06141=1187.802,-30.499,-42.955,179.793,5.699,149.070
C06142=1187.807,-30.749,-42.942,179.790,5.699,149.071
C06143=1187.812,-30.999,-42.930,179.788,5.698,149.072
C06144=1187.817,-31.248,-42.918,179.785,5.697,149.072
C06145=1187.823,-31.497,-42.905,179.783,5.697,149.073
C06146=1187.828,-31.747,-42.893,179.781,5.697,149.074
C06147=1187.832,-31.997,-42.880,179.779,5.696,149.074
C06148=1187.838,-32.246,-42.868,179.776,5.696,149.075
C06149=1187.843,-32.496,-42.856,179.773,5.696,149.075
C06150=1187.848,-32.746,-42.843,179.771,5.695,149.076
C06151=1187.853,-32.995,-42.831,179.769,5.695,149.077
C06152=1187.859,-33.245,-42.819,179.766,5.695,149.077
C06153=1187.864,-33.494,-42.806,179.764,5.694,149.078
C06154=1187.869,-33.744,-42.794,179.761,5.693,149.079
C06155=1187.874,-33.994,-42.781,179.759,5.694,149.079
C06156=1187.879,-34.244,-42.769,179.757,5.693,149.080
C06157=1187.884,-34.494,-42.757,179.754,5.693,149.081
C06158=1187.889,-34.743,-42.744,179.752,5.692,149.081
C06159=1187.895,-34.993,-42.732,179.749,5.692,149.082
C06160=1187.900,-35.242,-42.720,179.747,5.692,149.082
C06161=1187.905,-35.491,-42.707,179.745,5.691,149.083
C06162=1187.911,-35.741,-42.695,179.742,5.691,149.084
C06163=1187.916,-35.991,-42.683,179.740,5.690,149.084
C06164=1187.921,-36.241,-42.671,179.737,5.690,149.085
C06165=1187.926,-36.491,-42.658,179.735,5.690,149.086
C06166=1187.931,-36.741,-42.646,179.733,5.689,149.086
C06167=1187.936,-36.990,-42.633,179.730,5.689,149.087
C06168=1187.942,-37.240,-42.621,179.727,5.688,149.088
C06169=1187.946,-37.489,-42.609,179.725,5.689,149.088
C06170=1187.951,-37.739,-42.597,179.723,5.688,149.089
C06171=1187.957,-37.988,-42.585,179.721,5.687,149.089
C06172=1187.962,-38.238,-42.573,179.718,5.687,149.090
C06173=1187.967,-38.487,-42.560,179.716,5.687,149.091
C06174=1187.973,-38.737,-42.549,179.714,5.687,149.091
C06175=1187.978,-38.987,-42.537,179.711,5.686,149.092
C06176=1187.983,-39.237,-42.524,179.708,5.686,149.093
C06177=1187.988,-39.486,-42.513,179.706,5.685,149.093
C06178=1187.993,-39.735,-42.500,179.704,5.685,149.094
C06179=1187.998,-39.985,-42.488,179.701,5.685,149.095
C06180=1188.003,-40.235,-42.476,179.699,5.684,149.095
C06181=1188.009,-40.485,-42.464,179.696,5.684,149.096
C06182=1188.014,-40.735,-42.452,179.694,5.684,149.097
C06183=1188.019,-40.984,-42.439,179.692,5.683,149.097
C06184=1188.024,-41.234,-42.428,179.689,5.683,149.098
C06185=1188.029,-41.483,-42.415,179.686,5.682,149.099
C06186=1188.035,-41.733,-42.404,179.685,5.682,149.099
C06187=1188.040,-41.983,-42.392,179.682,5.682,149.100
C06188=1188.045,-42.232,-42.379,179.680,5.682,149.100
C06189=1188.050,-42.482,-42.368,179.677,5.681,149.101
C06190=1188.055,-42.732,-42.356,179.675,5.681,149.102
C06191=1188.060,-42.981,-42.343,179.673,5.681,149.102
C06192=1188.066,-43.231,-42.331,179.670,5.680,149.103
C06193=1188.071,-43.480,-42.320,179.667,5.680,149.104
C06194=1188.076,-43.730,-42.307,179.666,5.680,149.104
C06195=1188.081,-43.980,-42.296,179.663,5.679,149.105
C06196=1188.087,-44.230,-42.284,179.660,5.679,149.106
C06197=1188.091,-44.479,-42.272,179.658,5.678,149.106
C06198=1188.096,-44.729,-42.260,179.656,5.678,149.107
C06199=1188.102,-44.979,-42.248,179.653,5.678,149.108
C06200=1188.107,-45.228,-42.236,179.651,5.678,149.108
C06201=1188.112,-45.478,-42.225,179.649,5.677,149.109
C06202=1188.117,-45.727,-42.212,179.647,5.677,149.109
C06203=1188.123,-45.977,-42.200,179.644,5.677,149.110
C06204=1188.128,-46.227,-42.188,179.641,5.676,149.111
C06205=1188.133,-46.477,-42.177,179.639,5.675,149.111
C06206=1188.138,-46.726,-42.164,179.637,5.676,149.112
C06207=1188.143,-46.976,-42.153,179.634,5.675,149.113
C06208=1188.148,-47.226,-42.141,179.632,5.675,149.113
C06209=1188.154,-47.475,-42.130,179.630,5.675,149.114
C06210=1188.159,-47.725,-42.118,179.627,5.674,149.115
C06211=1188.164,-47.974,-42.106,179.625,5.674,149.115
C06212=1188.169,-48.224,-42.094,179.622,5.674,149.116
C06213=1188.175,-48.474,-42.082,179.620,5.673,149.116
C06214=1188.179,-48.723,-42.071,179.618,5.673,149.117
C06215=1188.185,-48.973,-42.059,179.615,5.673,149.118
C06216=1188.190,-49.244,-42.046,179.612,5.672,149.119
C06217=1188.196,-49.513,-42.033,179.610,5.672,149.119
C06218=1188.201,-49.784,-42.020,179.608,5.672,149.120
C06219=1188.207,-50.054,-42.009,179.605,5.672,149.121
C06220=1188.213,-50.304,-41.997,179.603,5.671,149.121
C06221=1188.218,-50.554,-41.985,179.600,5.670,149.122
C06222=1188.223,-50.803,-41.973,179.598,5.671,149.123
C06223=1188.228,-51.053,-41.961,179.595,5.670,149.123
C06224=1188.233,-51.303,-41.950,179.593,5.670,149.124
C06225=1188.238,-51.552,-41.938,179.591,5.669,149.124
C06226=1188.243,-51.802,-41.926,179.588,5.669,149.125
C06227=1188.249,-52.051,-41.915,179.586,5.669,149.126
C06228=1188.254,-52.301,-41.903,179.584,5.668,149.126
C06229=1188.259,-52.551,-41.892,179.582,5.669,149.127
C06230=1188.265,-52.801,-41.880,179.579,5.668,149.128
C06231=1188.269,-53.050,-41.869,179.577,5.667,149.128
C06232=1188.275,-53.300,-41.857,179.574,5.667,149.129
C06233=1188.279,-53.550,-41.845,179.572,5.667,149.130
C06234=1188.285,-53.799,-41.834,179.569,5.667,149.130
C06235=1188.291,-54.049,-41.822,179.567,5.666,149.131
C06236=1188.295,-54.299,-41.811,179.565,5.666,149.131
C06237=1188.301,-54.549,-41.799,179.562,5.666,149.132
C06238=1188.306,-54.798,-41.787,179.560,5.665,149.133
C06239=1188.311,-55.048,-41.776,179.558,5.665,149.133
C06240=1188.316,-55.297,-41.765,179.555,5.665,149.134
C06241=1188.322,-55.547,-41.753,179.553,5.665,149.135
C06242=1188.326,-55.797,-41.742,179.551,5.664,149.135
C06243=1188.332,-56.047,-41.730,179.548,5.664,149.136
C06244=1188.337,-56.296,-41.718,179.546,5.664,149.137
C06245=1188.343,-56.546,-41.707,179.543,5.663,149.137
C06246=1188.347,-56.795,-41.696,179.542,5.663,149.138
C06247=1188.353,-57.045,-41.684,179.539,5.663,149.139
C06248=1188.358,-57.295,-41.673,179.536,5.662,149.139
C06249=1188.362,-57.545,-41.662,179.535,5.662,149.140
C06250=1188.368,-57.794,-41.650,179.532,5.662,149.140
C06251=1188.373,-58.044,-41.639,179.529,5.662,149.141
C06252=1188.379,-58.294,-41.627,179.527,5.662,149.142
C06253=1188.383,-58.543,-41.616,179.525,5.661,149.142
C06254=1188.389,-58.793,-41.604,179.522,5.661,149.143
C06255=1188.394,-59.042,-41.593,179.520,5.660,149.144
C06256=1188.400,-59.293,-41.582,179.518,5.660,149.144
C06257=1188.404,-59.542,-41.571,179.515,5.660,149.145
C06258=1188.409,-59.792,-41.559,179.513,5.659,149.146
C06259=1188.415,-60.041,-41.548,179.511,5.660,149.146
C06260=1188.420,-60.291,-41.536,179.509,5.659,149.147
C06261=1188.425,-60.541,-41.525,179.506,5.658,149.147
C06262=1188.431,-60.790,-41.514,179.504,5.659,149.148
C06263=1188.436,-61.040,-41.503,179.501,5.658,149.149
C06264=1188.441,-61.290,-41.491,179.499,5.658,149.149
C06265=1188.446,-61.540,-41.480,179.497,5.658,149.150
C06266=1188.452,-61.789,-41.468,179.494,5.658,149.151
C06267=1188.457,-62.039,-41.458,179.492,5.657,149.151
C06268=1188.461,-62.289,-41.446,179.490,5.657,149.152
C06269=1188.467,-62.539,-41.435,179.487,5.657,149.153
C06270=1188.472,-62.788,-41.424,179.485,5.656,149.153
C06271=1188.477,-63.038,-41.413,179.483,5.656,149.154
C06272=1188.483,-63.288,-41.401,179.480,5.656,149.155
C06273=1188.488,-63.537,-41.390,179.478,5.655,149.155
C06274=1188.493,-63.787,-41.380,179.476,5.655,149.156
C06275=1188.498,-64.037,-41.368,179.473,5.655,149.156
C06276=1188.504,-64.286,-41.357,179.471,5.655,149.157
C06277=1188.508,-64.535,-41.346,179.469,5.655,149.158
C06278=1188.514,-64.786,-41.334,179.466,5.654,149.158
C06279=1188.519,-65.036,-41.323,179.464,5.654,149.159
C06280=1188.524,-65.285,-41.312,179.462,5.654,149.160
C06281=1188.530,-65.535,-41.301,179.460,5.653,149.160
C06282=1188.534,-65.785,-41.290,179.457,5.653,149.161
C06283=1188.540,-66.034,-41.279,179.455,5.653,149.162
C06284=1188.545,-66.284,-41.268,179.453,5.652,149.162
C06285=1188.550,-66.534,-41.256,179.450,5.652,149.163
C06286=1188.556,-66.783,-41.246,179.448,5.652,149.164
C06287=1188.560,-67.033,-41.235,179.445,5.652,149.164
C06288=1188.566,-67.282,-41.223,179.443,5.651,149.165
C06289=1188.571,-67.532,-41.213,179.441,5.651,149.165
C06290=1188.576,-67.782,-41.202,179.438,5.651,149.166
C06291=1188.582,-68.032,-41.191,179.436,5.650,149.167
C06292=1188.587,-68.282,-41.179,179.434,5.651,149.167
C06293=1188.592,-68.531,-41.168,179.431,5.650,149.168
C06294=1188.597,-68.781,-41.158,179.429,5.649,149.169
C06295=1188.603,-69.031,-41.146,179.427,5.650,149.169
C06296=1188.608,-69.280,-41.136,179.424,5.649,149.170
C06297=1188.613,-69.530,-41.125,179.422,5.650,149.171
C06298=1188.618,-69.780,-41.114,179.420,5.649,149.171
C06299=1188.623,-70.029,-41.103,179.417,5.648,149.172
C06300=1188.629,-70.280,-41.092,179.415,5.649,149.173
C06301=1188.634,-70.529,-41.081,179.413,5.648,149.173
C06302=1188.639,-70.778,-41.070,179.410,5.648,149.174
C06303=1188.644,-71.028,-41.059,179.408,5.648,149.174
C06304=1188.649,-71.277,-41.048,179.406,5.647,149.175
C06305=1188.655,-71.528,-41.037,179.404,5.647,149.176
C06306=1188.661,-71.777,-41.027,179.401,5.647,149.176
C06307=1188.665,-72.027,-41.015,179.399,5.647,149.177
C06308=1188.670,-72.277,-41.005,179.397,5.646,149.177
C06309=1188.676,-72.526,-40.994,179.395,5.646,149.178
C06310=1188.681,-72.777,-40.983,179.392,5.646,149.179
C06311=1188.687,-73.026,-40.972,179.390,5.646,149.179
C06312=1188.692,-73.276,-40.961,179.388,5.645,149.180
C06313=1188.697,-73.525,-40.950,179.385,5.645,149.181
C06314=1188.702,-73.775,-40.940,179.383,5.645,149.181
C06315=1188.707,-74.024,-40.929,179.381,5.645,149.182
C06316=1188.712,-74.274,-40.918,179.378,5.644,149.183
C06317=1188.718,-74.525,-40.907,179.376,5.644,149.183
C06318=1188.723,-74.774,-40.896,179.374,5.644,149.184
C06319=1188.728,-75.024,-40.886,179.372,5.644,149.185
C06320=1188.734,-75.294,-40.874,179.369,5.644,149.185
C06321=1188.740,-75.566,-40.863,179.366,5.643,149.186
C06322=1188.745,-75.837,-40.851,179.364,5.643,149.187
C06323=1188.751,-76.106,-40.839,179.362,5.643,149.187
C06324=1188.757,-76.357,-40.828,179.359,5.642,149.188
C06325=1188.762,-76.607,-40.818,179.357,5.642,149.189
C06326=1188.767,-76.856,-40.807,179.355,5.642,149.189
C06327=1188.773,-77.106,-40.796,179.352,5.642,149.190
C06328=1188.778,-77.356,-40.786,179.350,5.641,149.191
C06329=1188.783,-77.605,-40.775,179.348,5.642,149.191
C06330=1188.788,-77.855,-40.764,179.345,5.641,149.192
C06331=1188.793,-78.105,-40.754,179.343,5.641,149.192
C06332=1188.798,-78.354,-40.743,179.341,5.641,149.193
C06333=1188.804,-78.604,-40.733,179.339,5.640,149.194
C06334=1188.809,-78.854,-40.722,179.336,5.640,149.194
C06335=1188.814,-79.104,-40.712,179.334,5.640,149.195
C06336=1188.819,-79.353,-40.701,179.332,5.640,149.195
C06337=1188.825,-79.603,-40.690,179.329,5.640,149.196
C06338=1188.830,-79.853,-40.680,179.327,5.639,149.197
C06339=1188.835,-80.103,-40.670,179.325,5.639,149.197
C06340=1188.840,-80.352,-40.658,179.323,5.639,149.198
C06341=1188.845,-80.602,-40.648,179.320,5.638,149.199
C06342=1188.850,-80.852,-40.637,179.318,5.638,149.199
C06343=1188.856,-81.102,-40.627,179.316,5.638,149.200
C06344=1188.861,-81.350,-40.616,179.314,5.638,149.201
C06345=1188.866,-81.601,-40.606,179.311,5.637,149.201
C06346=1188.872,-81.850,-40.596,179.309,5.637,149.202
C06347=1188.877,-82.101,-40.585,179.307,5.637,149.203
C06348=1188.883,-82.350,-40.575,179.304,5.637,149.203
C06349=1188.887,-82.600,-40.563,179.302,5.637,149.204
C06350=1188.893,-82.849,-40.553,179.300,5.637,149.205
C06351=1188.898,-83.100,-40.543,179.297,5.636,149.205
C06352=1188.903,-83.349,-40.533,179.295,5.636,149.206
C06353=1188.909,-83.599,-40.522,179.293,5.636,149.206
C06354=1188.914,-83.849,-40.512,179.291,5.636,149.207
C06355=1188.919,-84.098,-40.501,179.288,5.635,149.208
C06356=1188.924,-84.348,-40.490,179.286,5.635,149.208
C06357=1188.930,-84.598,-40.480,179.284,5.635,149.209
C06358=1188.936,-84.847,-40.470,179.281,5.635,149.210
C06359=1188.940,-85.097,-40.460,179.279,5.635,149.210
C06360=1188.945,-85.347,-40.450,179.277,5.634,149.211
C06361=1188.950,-85.597,-40.439,179.275,5.635,149.211
C06362=1188.956,-85.846,-40.429,179.272,5.634,149.212
C06363=1188.962,-86.096,-40.419,179.270,5.633,149.213
C06364=1188.967,-86.346,-40.408,179.268,5.634,149.213
C06365=1188.972,-86.595,-40.397,179.266,5.633,149.214
C06366=1188.977,-86.845,-40.387,179.264,5.633,149.215
C06367=1188.982,-87.095,-40.377,179.261,5.633,149.215
C06368=1188.987,-87.344,-40.367,179.259,5.632,149.216
C06369=1188.992,-87.594,-40.356,179.257,5.632,149.216
C06370=1188.998,-87.844,-40.346,179.254,5.632,149.217
C06371=1189.003,-88.094,-40.335,179.252,5.632,149.218
C06372=1189.008,-88.344,-40.325,179.250,5.632,149.218
C06373=1189.014,-88.593,-40.315,179.248,5.632,149.219
C06374=1189.018,-88.843,-40.305,179.246,5.631,149.220
C06375=1189.024,-89.093,-40.295,179.243,5.631,149.220
C06376=1189.030,-89.342,-40.285,179.241,5.631,149.221
C06377=1189.035,-89.592,-40.274,179.239,5.630,149.221
C06378=1189.040,-89.842,-40.264,179.237,5.631,149.222
C06379=1189.045,-90.091,-40.254,179.234,5.630,149.223
C06380=1189.050,-90.341,-40.244,179.232,5.630,149.223
C06381=1189.056,-90.591,-40.233,179.230,5.630,149.224
C06382=1189.061,-90.841,-40.223,179.227,5.630,149.225
C06383=1189.066,-91.091,-40.213,179.226,5.630,149.225
C06384=1189.071,-91.340,-40.203,179.223,5.629,149.226
C06385=1189.077,-91.590,-40.193,179.221,5.630,149.227
C06386=1189.082,-91.840,-40.182,179.219,5.629,149.227
C06387=1189.088,-92.090,-40.173,179.216,5.628,149.228
C06388=1189.093,-92.340,-40.162,179.214,5.628,149.228
C06389=1189.097,-92.589,-40.153,179.212,5.628,149.229
C06390=1189.103,-92.839,-40.142,179.210,5.628,149.230
C06391=1189.109,-93.089,-40.132,179.207,5.628,149.230
C06392=1189.114,-93.338,-40.122,179.205,5.628,149.231
C06393=1189.118,-93.588,-40.112,179.203,5.628,149.232
C06394=1189.124,-93.838,-40.102,179.201,5.628,149.232
C06395=1189.130,-94.087,-40.091,179.198,5.627,149.233
C06396=1189.135,-94.338,-40.082,179.196,5.627,149.234
C06397=1189.140,-94.587,-40.072,179.194,5.627,149.234
C06398=1189.145,-94.837,-40.062,179.191,5.626,149.235
C06399=1189.151,-95.086,-40.052,179.190,5.626,149.235
C06400=1189.155,-95.336,-40.042,179.187,5.626,149.236
C06401=1189.161,-95.586,-40.031,179.185,5.626,149.237
C06402=1189.167,-95.836,-40.022,179.183,5.626,149.237
C06403=1189.172,-96.085,-40.012,179.180,5.625,149.238
C06404=1189.177,-96.335,-40.002,179.178,5.626,149.239
C06405=1189.182,-96.585,-39.992,179.176,5.625,149.239
C06406=1189.188,-96.835,-39.981,179.174,5.625,149.240
C06407=1189.193,-97.084,-39.972,179.172,5.624,149.240
C06408=1189.198,-97.335,-39.962,179.170,5.625,149.241
C06409=1189.204,-97.584,-39.952,179.167,5.624,149.242
C06410=1189.208,-97.833,-39.942,179.165,5.624,149.242
C06411=1189.214,-98.083,-39.932,179.163,5.624,149.243
C06412=1189.219,-98.334,-39.922,179.161,5.624,149.243
C06413=1189.224,-98.583,-39.912,179.158,5.624,149.244
C06414=1189.230,-98.833,-39.902,179.156,5.623,149.245
C06415=1189.236,-99.083,-39.893,179.154,5.623,149.245
C06416=1189.241,-99.332,-39.883,179.151,5.623,149.246
C06417=1189.246,-99.582,-39.872,179.149,5.623,149.247
C06418=1189.250,-99.831,-39.863,179.147,5.622,149.247
C06419=1189.256,-100.082,-39.853,179.145,5.623,149.248
C06420=1189.262,-100.331,-39.843,179.143,5.622,149.248
C06421=1189.267,-100.580,-39.834,179.141,5.622,149.249
C06422=1189.272,-100.831,-39.824,179.138,5.622,149.250
C06423=1189.277,-101.080,-39.814,179.136,5.622,149.250
C06424=1189.283,-101.352,-39.803,179.134,5.622,149.251
C06425=1189.289,-101.623,-39.793,179.131,5.621,149.252
C06426=1189.294,-101.895,-39.782,179.129,5.622,149.252
C06427=1189.300,-102.167,-39.771,179.126,5.621,149.253
C06428=1189.305,-102.416,-39.761,179.124,5.620,149.254
C06429=1189.311,-102.666,-39.752,179.122,5.621,149.254
C06430=1189.316,-102.915,-39.742,179.120,5.620,149.255
C06431=1189.321,-103.166,-39.732,179.118,5.620,149.256
C06432=1189.326,-103.416,-39.723,179.115,5.620,149.256
C06433=1189.332,-103.665,-39.712,179.114,5.620,149.257
C06434=1189.338,-103.915,-39.703,179.111,5.620,149.257
C06435=1189.343,-104.164,-39.693,179.109,5.620,149.258
C06436=1189.348,-104.415,-39.684,179.107,5.619,149.259
C06437=1189.353,-104.664,-39.674,179.105,5.619,149.259
C06438=1189.358,-104.914,-39.664,179.102,5.619,149.260
C06439=1189.363,-105.164,-39.655,179.100,5.618,149.261
C06440=1189.369,-105.414,-39.645,179.098,5.618,149.261
C06441=1189.374,-105.663,-39.636,179.095,5.618,149.262
C06442=1189.380,-105.913,-39.625,179.094,5.618,149.262
C06443=1189.385,-106.163,-39.617,179.091,5.618,149.263
C06444=1189.391,-106.412,-39.606,179.089,5.618,149.264
C06445=1189.395,-106.663,-39.597,179.087,5.617,149.264
C06446=1189.401,-106.912,-39.587,179.085,5.618,149.265
C06447=1189.406,-107.162,-39.577,179.083,5.617,149.265
C06448=1189.412,-107.412,-39.568,179.080,5.617,149.266
C06449=1189.416,-107.661,-39.558,179.078,5.617,149.267
C06450=1189.422,-107.911,-39.549,179.076,5.617,149.267
C06451=1189.427,-108.160,-39.539,179.073,5.617,149.268
C06452=1189.432,-108.410,-39.530,179.072,5.617,149.268
C06453=1189.438,-108.660,-39.521,179.069,5.616,149.269
C06454=1189.443,-108.910,-39.511,179.068,5.616,149.270
C06455=1189.448,-109.161,-39.501,179.065,5.616,149.270
C06456=1189.453,-109.410,-39.492,179.063,5.616,149.271
C06457=1189.459,-109.660,-39.482,179.061,5.615,149.272
C06458=1189.464,-109.909,-39.472,179.059,5.616,149.272
C06459=1189.470,-110.159,-39.463,179.056,5.615,149.273
C06460=1189.475,-110.409,-39.453,179.054,5.615,149.273
C06461=1189.480,-110.658,-39.444,179.052,5.615,149.274
C06462=1189.486,-110.909,-39.435,179.050,5.615,149.275
C06463=1189.491,-111.158,-39.425,179.047,5.615,149.275
C06464=1189.497,-111.408,-39.416,179.045,5.614,149.276
C06465=1189.501,-111.657,-39.406,179.043,5.614,149.277
C06466=1189.507,-111.907,-39.397,179.041,5.613,149.277
C06467=1189.513,-112.157,-39.388,179.039,5.614,149.278
C06468=1189.517,-112.406,-39.378,179.037,5.613,149.278
C06469=1189.523,-112.657,-39.369,179.034,5.614,149.279
C06470=1189.528,-112.906,-39.359,179.032,5.613,149.279
C06471=1189.533,-113.156,-39.350,179.030,5.613,149.280
C06472=1189.539,-113.407,-39.340,179.028,5.613,149.281
C06473=1189.544,-113.656,-39.331,179.026,5.613,149.281
C06474=1189.549,-113.906,-39.322,179.023,5.612,149.282
C06475=1189.555,-114.156,-39.312,179.022,5.612,149.283
C06476=1189.559,-114.405,-39.303,179.019,5.612,149.283
C06477=1189.565,-114.655,-39.294,179.017,5.612,149.284
C06478=1189.571,-114.905,-39.284,179.015,5.612,149.285
C06479=1189.575,-115.154,-39.275,179.013,5.612,149.285
C06480=1189.581,-115.404,-39.266,179.010,5.611,149.286
C06481=1189.586,-115.654,-39.256,179.008,5.612,149.286
C06482=1189.592,-115.904,-39.248,179.006,5.611,149.287
C06483=1189.596,-116.153,-39.238,179.004,5.611,149.288
C06484=1189.602,-116.404,-39.228,179.002,5.610,149.288
C06485=1189.608,-116.653,-39.219,179.000,5.611,149.289
C06486=1189.612,-116.903,-39.210,178.998,5.610,149.289
C06487=1189.618,-117.153,-39.200,178.996,5.611,149.290
C06488=1189.623,-117.403,-39.191,178.993,5.610,149.291
C06489=1189.629,-117.652,-39.183,178.991,5.610,149.291
C06490=1189.634,-117.901,-39.173,178.989,5.609,149.292
C06491=1189.640,-118.151,-39.164,178.987,5.610,149.292
C06492=1189.645,-118.401,-39.155,178.985,5.609,149.293
C06493=1189.650,-118.651,-39.146,178.983,5.609,149.294
C06494=1189.656,-118.901,-39.137,178.981,5.610,149.294
C06495=1189.661,-119.150,-39.127,178.978,5.609,149.295
C06496=1189.666,-119.400,-39.118,178.976,5.609,149.296
C06497=1189.671,-119.650,-39.109,178.974,5.609,149.296
C06498=1189.677,-119.900,-39.100,178.972,5.609,149.297
C06499=1189.683,-120.150,-39.091,178.970,5.608,149.297
C06500=1189.687,-120.399,-39.081,178.968,5.609,149.298
C06501=1189.693,-120.649,-39.072,178.966,5.608,149.298
C06502=1189.698,-120.899,-39.063,178.963,5.608,149.299
C06503=1189.703,-121.149,-39.054,178.961,5.608,149.300
C06504=1189.709,-121.399,-39.045,178.959,5.608,149.300
C06505=1189.714,-121.649,-39.036,178.957,5.607,149.301
C06506=1189.719,-121.899,-39.027,178.955,5.608,149.302
C06507=1189.724,-122.148,-39.018,178.953,5.607,149.302
C06508=1189.729,-122.398,-39.009,178.951,5.607,149.303
C06509=1189.736,-122.647,-39.000,178.948,5.606,149.303
C06510=1189.741,-122.897,-38.991,178.946,5.607,149.304
C06511=1189.746,-123.147,-38.982,178.944,5.606,149.304
C06512=1189.751,-123.397,-38.973,178.942,5.606,149.305
C06513=1189.756,-123.647,-38.964,178.940,5.606,149.306
C06514=1189.762,-123.897,-38.954,178.938,5.606,149.306
C06515=1189.767,-124.147,-38.946,178.936,5.605,149.307
C06516=1189.773,-124.396,-38.937,178.934,5.606,149.308
C06517=1189.777,-124.646,-38.927,178.931,5.605,149.308
C06518=1189.783,-124.896,-38.918,178.929,5.605,149.309
C06519=1189.788,-125.145,-38.910,178.927,5.605,149.309
C06520=1189.794,-125.395,-38.901,178.925,5.605,149.310
C06521=1189.799,-125.645,-38.891,178.923,5.605,149.310
C06522=1189.805,-125.895,-38.882,178.921,5.605,149.311
C06523=1189.810,-126.144,-38.873,178.919,5.605,149.312
C06524=1189.815,-126.394,-38.865,178.916,5.604,149.312
C06525=1189.820,-126.644,-38.856,178.915,5.604,149.313
C06526=1189.825,-126.894,-38.847,178.912,5.604,149.314
C06527=1189.831,-127.143,-38.838,178.911,5.604,149.314
C06528=1189.410,-127.155,-38.878,178.906,5.608,149.316
C06529=1189.405,-126.905,-38.887,178.908,5.607,149.315
C06530=1189.400,-126.655,-38.895,178.910,5.608,149.315
C06531=1189.394,-126.406,-38.904,178.912,5.608,149.314
C06532=1189.388,-126.156,-38.913,178.915,5.608,149.314
C06533=1189.383,-125.906,-38.922,178.917,5.608,149.313
C06534=1189.378,-125.656,-38.931,178.919,5.609,149.313
C06535=1189.373,-125.406,-38.940,178.921,5.608,149.312
C06536=1189.367,-125.156,-38.949,178.923,5.609,149.311
C06537=1189.362,-124.906,-38.958,178.925,5.609,149.311
C06538=1189.357,-124.657,-38.967,178.928,5.609,149.310
C06539=1189.351,-124.407,-38.975,178.930,5.609,149.309
C06540=1189.345,-124.157,-38.985,178.931,5.609,149.309
C06541=1189.340,-123.907,-38.994,178.934,5.609,149.308
C06542=1189.335,-123.658,-39.003,178.935,5.609,149.308
C06543=1189.330,-123.408,-39.012,178.938,5.610,149.307
C06544=1189.325,-123.158,-39.020,178.940,5.610,149.307
C06545=1189.320,-122.908,-39.029,178.942,5.610,149.306
C06546=1189.314,-122.658,-39.039,178.944,5.610,149.305
C06547=1189.309,-122.409,-39.048,178.947,5.610,149.305
C06548=1189.304,-122.159,-39.057,178.948,5.610,149.304
C06549=1189.298,-121.910,-39.066,178.951,5.611,149.303
C06550=1189.293,-121.660,-39.075,178.953,5.611,149.303
C06551=1189.287,-121.410,-39.084,178.955,5.611,149.302
C06552=1189.282,-121.160,-39.093,178.957,5.611,149.302
C06553=1189.276,-120.910,-39.102,178.960,5.612,149.301
C06554=1189.271,-120.660,-39.111,178.962,5.611,149.300
C06555=1189.266,-120.411,-39.121,178.964,5.612,149.300
C06556=1189.260,-120.161,-39.130,178.966,5.611,149.299
C06557=1189.255,-119.911,-39.139,178.968,5.612,149.299
C06558=1189.250,-119.661,-39.148,178.970,5.612,149.298
C06559=1189.245,-119.411,-39.157,178.972,5.613,149.297
C06560=1189.239,-119.162,-39.167,178.974,5.612,149.297
C06561=1189.234,-118.912,-39.176,178.977,5.613,149.296
C06562=1189.229,-118.662,-39.185,178.979,5.613,149.295
C06563=1189.224,-118.412,-39.194,178.981,5.613,149.295
C06564=1189.218,-118.162,-39.203,178.983,5.613,149.294
C06565=1189.213,-117.913,-39.213,178.985,5.614,149.294
C06566=1189.208,-117.663,-39.222,178.987,5.613,149.293
C06567=1189.203,-117.413,-39.231,178.990,5.614,149.293
C06568=1189.197,-117.163,-39.240,178.992,5.614,149.292
C06569=1189.192,-116.914,-39.250,178.994,5.615,149.291
C06570=1189.186,-116.664,-39.258,178.996,5.614,149.291
C06571=1189.180,-116.414,-39.268,178.999,5.614,149.290
C06572=1189.175,-116.164,-39.277,179.000,5.614,149.289
C06573=1189.170,-115.915,-39.286,179.003,5.615,149.289
C06574=1189.164,-115.665,-39.296,179.004,5.615,149.288
C06575=1189.159,-115.415,-39.305,179.007,5.615,149.288
C06576=1189.154,-115.165,-39.314,179.009,5.615,149.287
C06577=1189.149,-114.916,-39.323,179.011,5.616,149.286
C06578=1189.143,-114.666,-39.333,179.013,5.616,149.286
C06579=1189.138,-114.416,-39.342,179.016,5.616,149.285
C06580=1189.133,-114.166,-39.352,179.017,5.616,149.285
C06581=1189.127,-113.917,-39.361,179.020,5.616,149.284
C06582=1189.122,-113.667,-39.370,179.022,5.616,149.283
C06583=1189.117,-113.417,-39.380,179.024,5.617,149.283
C06584=1189.112,-113.167,-39.389,179.026,5.616,149.282
C06585=1189.107,-112.917,-39.398,179.028,5.617,149.282
C06586=1189.101,-112.667,-39.408,179.031,5.617,149.281
C06587=1189.096,-112.417,-39.417,179.033,5.617,149.280
C06588=1189.091,-112.168,-39.427,179.035,5.617,149.280
C06589=1189.085,-111.918,-39.436,179.037,5.618,149.279
C06590=1189.080,-111.668,-39.445,179.039,5.617,149.278
C06591=1189.075,-111.419,-39.455,179.041,5.618,149.278
C06592=1189.069,-111.169,-39.464,179.043,5.618,149.277
C06593=1189.064,-110.919,-39.473,179.046,5.618,149.277
C06594=1189.059,-110.669,-39.483,179.048,5.618,149.276
C06595=1189.054,-110.420,-39.492,179.050,5.619,149.275
C06596=1189.048,-110.170,-39.502,179.052,5.619,149.275
C06597=1189.043,-109.920,-39.511,179.055,5.619,149.274
C06598=1189.038,-109.671,-39.521,179.056,5.619,149.274
C06599=1189.032,-109.421,-39.530,179.059,5.619,149.273
C06600=1189.027,-109.172,-39.540,179.061,5.619,149.272
C06601=1189.022,-108.921,-39.550,179.063,5.620,149.272
C06602=1189.017,-108.671,-39.559,179.065,5.619,149.271
C06603=1189.011,-108.421,-39.569,179.067,5.620,149.271
C06604=1189.006,-108.171,-39.578,179.070,5.620,149.270
C06605=1189.000,-107.922,-39.588,179.072,5.621,149.269
C06606=1188.995,-107.672,-39.597,179.074,5.620,149.269
C06607=1188.990,-107.423,-39.607,179.077,5.621,149.268
C06608=1188.984,-107.173,-39.616,179.078,5.621,149.267
C06609=1188.980,-106.923,-39.626,179.081,5.621,149.267
C06610=1188.974,-106.673,-39.635,179.082,5.621,149.266
C06611=1188.969,-106.423,-39.645,179.085,5.621,149.266
C06612=1188.963,-106.173,-39.655,179.087,5.622,149.265
C06613=1188.959,-105.924,-39.664,179.089,5.622,149.264
C06614=1188.953,-105.674,-39.674,179.092,5.622,149.264
C06615=1188.948,-105.424,-39.683,179.094,5.622,149.263
C06616=1188.942,-105.175,-39.694,179.096,5.622,149.262
C06617=1188.937,-104.925,-39.702,179.098,5.622,149.262
C06618=1188.931,-104.676,-39.713,179.101,5.623,149.261
C06619=1188.927,-104.425,-39.722,179.103,5.622,149.260
C06620=1188.921,-104.175,-39.732,179.105,5.623,149.260
C06621=1188.916,-103.926,-39.742,179.107,5.623,149.259
C06622=1188.911,-103.676,-39.751,179.109,5.624,149.259
C06623=1188.905,-103.427,-39.761,179.111,5.623,149.258
C06624=1188.900,-103.177,-39.770,179.114,5.624,149.257
C06625=1188.895,-102.926,-39.781,179.115,5.624,149.257
C06626=1188.890,-102.677,-39.791,179.118,5.624,149.256
C06627=1188.884,-102.427,-39.800,179.120,5.624,149.256
C06628=1188.879,-102.178,-39.810,179.122,5.624,149.255
C06629=1188.873,-101.906,-39.820,179.125,5.625,149.254
C06630=1188.868,-101.634,-39.831,179.127,5.624,149.254
C06631=1188.862,-101.363,-39.841,179.129,5.625,149.253
C06632=1188.856,-101.091,-39.853,179.132,5.626,149.252
C06633=1188.851,-100.842,-39.862,179.134,5.625,149.252
C06634=1188.845,-100.592,-39.872,179.136,5.626,149.251
C06635=1188.841,-100.342,-39.882,179.138,5.626,149.250
C06636=1188.835,-100.092,-39.891,179.141,5.626,149.250
C06637=1188.829,-99.842,-39.902,179.143,5.626,149.249
C06638=1188.824,-99.593,-39.911,179.145,5.626,149.249
C06639=1188.819,-99.343,-39.922,179.148,5.627,149.248
C06640=1188.814,-99.093,-39.931,179.150,5.627,149.247
C06641=1188.809,-98.844,-39.941,179.152,5.627,149.247
C06642=1188.803,-98.594,-39.951,179.154,5.627,149.246
C06643=1188.798,-98.344,-39.960,179.157,5.628,149.245
C06644=1188.793,-98.094,-39.971,179.159,5.627,149.245
C06645=1188.787,-97.844,-39.981,179.161,5.628,149.244
C06646=1188.782,-97.595,-39.990,179.163,5.628,149.244
C06647=1188.776,-97.345,-40.000,179.165,5.628,149.243
C06648=1188.771,-97.095,-40.010,179.167,5.628,149.242
C06649=1188.767,-96.845,-40.020,179.170,5.628,149.242
C06650=1188.761,-96.596,-40.030,179.172,5.629,149.241
C06651=1188.755,-96.346,-40.040,179.174,5.629,149.240
C06652=1188.750,-96.097,-40.049,179.176,5.630,149.240
C06653=1188.745,-95.846,-40.060,179.178,5.629,149.239
C06654=1188.740,-95.597,-40.070,179.181,5.630,149.239
C06655=1188.735,-95.348,-40.080,179.183,5.630,149.238
C06656=1188.729,-95.098,-40.090,179.185,5.630,149.237
C06657=1188.724,-94.847,-40.100,179.187,5.630,149.237
C06658=1188.718,-94.598,-40.110,179.190,5.630,149.236
C06659=1188.713,-94.348,-40.120,179.192,5.631,149.235
C06660=1188.708,-94.098,-40.130,179.194,5.631,149.235
C06661=1188.703,-93.849,-40.140,179.197,5.631,149.234
C06662=1188.697,-93.599,-40.151,179.199,5.631,149.234
C06663=1188.692,-93.350,-40.160,179.201,5.632,149.233
C06664=1188.687,-93.099,-40.170,179.203,5.631,149.232
C06665=1188.681,-92.849,-40.180,179.206,5.632,149.232
C06666=1188.676,-92.600,-40.191,179.208,5.632,149.231
C06667=1188.672,-92.350,-40.201,179.210,5.632,149.230
C06668=1188.666,-92.100,-40.211,179.212,5.633,149.230
C06669=1188.660,-91.851,-40.221,179.214,5.632,149.229
C06670=1188.655,-91.601,-40.232,179.217,5.633,149.228
C06671=1188.651,-91.351,-40.241,179.218,5.633,149.228
C06672=1188.645,-91.102,-40.251,179.221,5.633,149.227
C06673=1188.639,-90.852,-40.262,179.224,5.634,149.227
C06674=1188.634,-90.602,-40.272,179.225,5.634,149.226
C06675=1188.629,-90.352,-40.282,179.228,5.634,149.225
C06676=1188.624,-90.103,-40.292,179.230,5.634,149.225
C06677=1188.619,-89.853,-40.303,179.232,5.634,149.224
C06678=1188.613,-89.603,-40.313,179.234,5.634,149.223
C06679=1188.608,-89.354,-40.323,179.237,5.635,149.223
C06680=1188.603,-89.104,-40.334,179.239,5.635,149.222
C06681=1188.598,-88.854,-40.343,179.241,5.635,149.222
C06682=1188.593,-88.604,-40.354,179.244,5.636,149.221
C06683=1188.587,-88.355,-40.364,179.246,5.635,149.220
C06684=1188.582,-88.105,-40.374,179.248,5.636,149.220
C06685=1188.577,-87.855,-40.385,179.250,5.636,149.219
C06686=1188.571,-87.605,-40.395,179.253,5.636,149.218
C06687=1188.566,-87.356,-40.405,179.255,5.636,149.218
C06688=1188.561,-87.106,-40.415,179.257,5.636,149.217
C06689=1188.556,-86.856,-40.425,179.260,5.637,149.217
C06690=1188.550,-86.607,-40.436,179.262,5.636,149.216
C06691=1188.545,-86.356,-40.446,179.264,5.637,149.215
C06692=1188.539,-86.107,-40.456,179.266,5.638,149.215
C06693=1188.534,-85.857,-40.467,179.269,5.637,149.214
C06694=1188.529,-85.607,-40.477,179.271,5.638,149.213
C06695=1188.524,-85.358,-40.487,179.273,5.638,149.213
C06696=1188.519,-85.108,-40.497,179.275,5.638,149.212
C06697=1188.513,-84.858,-40.507,179.278,5.639,149.212
C06698=1188.509,-84.609,-40.519,179.280,5.638,149.211
C06699=1188.503,-84.359,-40.529,179.282,5.639,149.210
C06700=1188.497,-84.109,-40.539,179.284,5.639,149.210
C06701=1188.492,-83.859,-40.550,179.287,5.639,149.209
C06702=1188.487,-83.610,-40.560,179.288,5.639,149.209
C06703=1188.482,-83.359,-40.571,179.291,5.640,149.208
C06704=1188.476,-83.110,-40.581,179.294,5.640,149.207
C06705=1188.472,-82.860,-40.592,179.295,5.640,149.207
C06706=1188.466,-82.611,-40.602,179.298,5.641,149.206
C06707=1188.460,-82.361,-40.612,179.300,5.640,149.205
C06708=1188.456,-82.111,-40.622,179.302,5.641,149.205
C06709=1188.450,-81.862,-40.633,179.305,5.641,149.204
C06710=1188.446,-81.612,-40.644,179.307,5.641,149.203
C06711=1188.440,-81.362,-40.654,179.309,5.642,149.203
C06712=1188.435,-81.112,-40.665,179.312,5.642,149.202
C06713=1188.430,-80.863,-40.675,179.314,5.642,149.201
C06714=1188.425,-80.612,-40.685,179.316,5.643,149.201
C06715=1188.419,-80.364,-40.696,179.318,5.642,149.200
C06716=1188.414,-80.113,-40.707,179.321,5.643,149.199
C06717=1188.409,-79.864,-40.717,179.323,5.643,149.199
C06718=1188.403,-79.614,-40.727,179.325,5.643,149.198
C06719=1188.398,-79.365,-40.739,179.328,5.643,149.198
C06720=1188.393,-79.115,-40.749,179.329,5.643,149.197
C06721=1188.388,-78.865,-40.759,179.332,5.644,149.196
C06722=1188.382,-78.615,-40.770,179.335,5.644,149.196
C06723=1188.378,-78.366,-40.781,179.336,5.644,149.195
C06724=1188.371,-78.116,-40.792,179.339,5.645,149.194
C06725=1188.366,-77.866,-40.802,179.341,5.644,149.194
C06726=1188.361,-77.617,-40.813,179.344,5.645,149.193
C06727=1188.356,-77.366,-40.824,179.346,5.646,149.193
C06728=1188.350,-77.117,-40.834,179.348,5.645,149.192
C06729=1188.346,-76.867,-40.845,179.351,5.646,149.191
C06730=1188.340,-76.618,-40.856,179.353,5.646,149.191
C06731=1188.335,-76.367,-40.866,179.355,5.646,149.190
C06732=1188.330,-76.118,-40.877,179.358,5.646,149.189
C06733=1188.324,-75.847,-40.889,179.360,5.647,149.189
C06734=1188.319,-75.576,-40.900,179.362,5.647,149.188
C06735=1188.312,-75.305,-40.911,179.365,5.647,149.187
C06736=1188.307,-75.034,-40.924,179.367,5.648,149.187
C06737=1188.301,-74.785,-40.934,179.369,5.647,149.186
C06738=1188.297,-74.535,-40.945,179.372,5.648,149.185
C06739=1188.292,-74.285,-40.956,179.374,5.649,149.185
C06740=1188.286,-74.036,-40.967,179.376,5.648,149.184
C06741=1188.281,-73.786,-40.977,179.379,5.649,149.183
C06742=1188.275,-73.536,-40.988,179.381,5.649,149.183
C06743=1188.270,-73.286,-40.999,179.383,5.649,149.182
C06744=1188.265,-73.037,-41.010,179.386,5.649,149.181
C06745=1188.260,-72.787,-41.021,179.388,5.650,149.181
C06746=1188.254,-72.538,-41.031,179.390,5.650,149.180
C06747=1188.250,-72.288,-41.042,179.393,5.650,149.180
C06748=1188.244,-72.037,-41.054,179.394,5.650,149.179
C06749=1188.239,-71.788,-41.064,179.397,5.651,149.178
C06750=1188.234,-71.538,-41.075,179.400,5.651,149.178
C06751=1188.228,-71.289,-41.086,179.402,5.651,149.177
C06752=1188.223,-71.039,-41.097,179.404,5.652,149.176
C06753=1188.218,-70.789,-41.107,179.407,5.652,149.176
C06754=1188.212,-70.540,-41.119,179.409,5.652,149.175
C06755=1188.208,-70.290,-41.130,179.411,5.652,149.175
C06756=1188.202,-70.040,-41.140,179.414,5.653,149.174
C06757=1188.197,-69.791,-41.151,179.416,5.652,149.173
C06758=1188.191,-69.541,-41.162,179.418,5.653,149.173
C06759=1188.186,-69.291,-41.173,179.420,5.653,149.172
C06760=1188.181,-69.041,-41.184,179.423,5.653,149.171
C06761=1188.176,-68.792,-41.195,179.425,5.654,149.171
C06762=1188.171,-68.542,-41.206,179.427,5.654,149.170
C06763=1188.166,-68.292,-41.217,179.430,5.654,149.169
C06764=1188.160,-68.042,-41.228,179.432,5.655,149.169
C06765=1188.155,-67.793,-41.239,179.434,5.655,149.168
C06766=1188.150,-67.544,-41.250,179.436,5.655,149.168
C06767=1188.144,-67.293,-41.261,179.439,5.655,149.167
C06768=1188.140,-67.044,-41.272,179.441,5.655,149.166
C06769=1188.134,-66.794,-41.283,179.443,5.656,149.166
C06770=1188.128,-66.544,-41.294,179.446,5.656,149.165
C06771=1188.124,-66.295,-41.306,179.448,5.656,149.164
C06772=1188.118,-66.045,-41.316,179.450,5.657,149.164
C06773=1188.114,-65.795,-41.327,179.453,5.657,149.163
C06774=1188.108,-65.545,-41.339,179.455,5.657,149.162
C06775=1188.102,-65.296,-41.349,179.457,5.658,149.162
C06776=1188.098,-65.046,-41.361,179.460,5.658,149.161
C06777=1188.092,-64.796,-41.372,179.462,5.658,149.160
C06778=1188.087,-64.547,-41.383,179.464,5.658,149.160
C06779=1188.082,-64.297,-41.394,179.467,5.659,149.159
C06780=1188.077,-64.047,-41.406,179.469,5.658,149.159
C06781=1188.071,-63.798,-41.416,179.472,5.659,149.158
C06782=1188.066,-63.548,-41.427,179.474,5.660,149.157
C06783=1188.061,-63.298,-41.439,179.476,5.659,149.157
C06784=1188.056,-63.049,-41.450,179.479,5.660,149.156
C06785=1188.051,-62.799,-41.461,179.481,5.661,149.155
C06786=1188.045,-62.549,-41.473,179.483,5.660,149.155
C06787=1188.041,-62.299,-41.484,179.486,5.661,149.154
C06788=1188.035,-62.050,-41.495,179.488,5.661,149.153
C06789=1188.029,-61.800,-41.506,179.490,5.661,149.153
C06790=1188.025,-61.550,-41.517,179.492,5.661,149.152
C06791=1188.019,-61.301,-41.529,179.495,5.662,149.151
C06792=1188.014,-61.051,-41.540,179.497,5.662,149.151
C06793=1188.009,-60.801,-41.551,179.499,5.662,149.150
C06794=1188.004,-60.551,-41.563,179.502,5.663,149.150
C06795=1187.998,-60.302,-41.573,179.504,5.663,149.149
C06796=1187.993,-60.052,-41.585,179.506,5.663,149.148
C06797=1187.988,-59.803,-41.597,179.509,5.664,149.148
C06798=1187.983,-59.553,-41.607,179.511,5.663,149.147
C06799=1187.977,-59.303,-41.619,179.513,5.664,149.146
C06800=1187.973,-59.054,-41.630,179.516,5.665,149.146
C06801=1187.967,-58.804,-41.642,179.518,5.664,149.145
C06802=1187.962,-58.554,-41.653,179.521,5.665,149.144
C06803=1187.957,-58.305,-41.664,179.523,5.665,149.144
C06804=1187.952,-58.055,-41.676,179.525,5.666,149.143
C06805=1187.947,-57.805,-41.687,179.528,5.665,149.142
C06806=1187.941,-57.555,-41.699,179.530,5.666,149.142
C06807=1187.937,-57.305,-41.710,179.532,5.667,149.141
C06808=1187.931,-57.056,-41.721,179.534,5.666,149.141
C06809=1187.926,-56.807,-41.733,179.537,5.667,149.140
C06810=1187.920,-56.557,-41.744,179.539,5.668,149.139
C06811=1187.916,-56.307,-41.756,179.541,5.667,149.139
C06812=1187.910,-56.057,-41.768,179.544,5.668,149.138
C06813=1187.905,-55.808,-41.779,179.546,5.668,149.138
C06814=1187.900,-55.558,-41.790,179.548,5.668,149.137
C06815=1187.895,-55.309,-41.802,179.551,5.669,149.136
C06816=1187.889,-55.059,-41.814,179.554,5.669,149.135
C06817=1187.885,-54.809,-41.825,179.556,5.670,149.135
C06818=1187.879,-54.560,-41.836,179.558,5.669,149.134
C06819=1187.874,-54.310,-41.847,179.561,5.670,149.134
C06820=1187.868,-54.060,-41.859,179.563,5.671,149.133
C06821=1187.864,-53.810,-41.870,179.565,5.670,149.132
C06822=1187.858,-53.560,-41.882,179.568,5.671,149.132
C06823=1187.853,-53.310,-41.893,179.570,5.671,149.131
C06824=1187.848,-53.061,-41.906,179.572,5.672,149.130
C06825=1187.843,-52.812,-41.917,179.574,5.672,149.130
C06826=1187.838,-52.562,-41.929,179.577,5.672,149.129
C06827=1187.832,-52.312,-41.941,179.580,5.672,149.128
C06828=1187.828,-52.063,-41.952,179.581,5.673,149.128
C06829=1187.822,-51.813,-41.964,179.584,5.673,149.127
C06830=1187.817,-51.563,-41.975,179.587,5.673,149.126
C06831=1187.811,-51.314,-41.987,179.589,5.674,149.126
C06832=1187.806,-51.064,-41.999,179.591,5.674,149.125
C06833=1187.801,-50.814,-42.010,179.594,5.674,149.125
C06834=1187.796,-50.564,-42.022,179.596,5.675,149.124
C06835=1187.791,-50.315,-42.033,179.598,5.675,149.123
C06836=1187.786,-50.065,-42.045,179.601,5.675,149.123
C06837=1187.780,-49.795,-42.057,179.603,5.676,149.122
C06838=1187.774,-49.525,-42.070,179.606,5.676,149.121
C06839=1187.769,-49.254,-42.083,179.609,5.676,149.121
C06840=1187.763,-48.984,-42.095,179.611,5.677,149.120
C06841=1187.758,-48.734,-42.107,179.613,5.677,149.119
C06842=1187.753,-48.485,-42.119,179.616,5.677,149.119
C06843=1187.748,-48.235,-42.131,179.618,5.678,149.118
C06844=1187.742,-47.985,-42.143,179.621,5.678,149.117
C06845=1187.738,-47.736,-42.154,179.623,5.678,149.117
C06846=1187.732,-47.486,-42.166,179.625,5.679,149.116
C06847=1187.727,-47.236,-42.178,179.628,5.679,149.115
C06848=1187.722,-46.987,-42.190,179.630,5.679,149.115
C06849=1187.717,-46.737,-42.202,179.633,5.679,149.114
C06850=1187.711,-46.488,-42.213,179.635,5.680,149.114
C06851=1187.705,-46.238,-42.225,179.637,5.680,149.113
C06852=1187.701,-45.989,-42.237,179.639,5.680,149.112
C06853=1187.696,-45.739,-42.249,179.642,5.681,149.112
C06854=1187.690,-45.489,-42.261,179.644,5.681,149.111
C06855=1187.686,-45.239,-42.272,179.647,5.682,149.110
C06856=1187.680,-44.989,-42.284,179.649,5.681,149.110
C06857=1187.675,-44.740,-42.297,179.651,5.682,149.109
C06858=1187.670,-44.490,-42.309,179.654,5.683,149.108
C06859=1187.665,-44.240,-42.320,179.657,5.683,149.108
C06860=1187.660,-43.991,-42.333,179.659,5.683,149.107
C06861=1187.654,-43.741,-42.345,179.661,5.684,149.107
C06862=1187.649,-43.491,-42.356,179.663,5.684,149.106
C06863=1187.644,-43.242,-42.368,179.666,5.684,149.105
C06864=1187.639,-42.992,-42.380,179.668,5.684,149.104
C06865=1187.634,-42.742,-42.392,179.670,5.685,149.104
C06866=1187.628,-42.492,-42.404,179.673,5.685,149.103
C06867=1187.623,-42.243,-42.417,179.676,5.686,149.103
C06868=1187.618,-41.993,-42.428,179.678,5.685,149.102
C06869=1187.613,-41.744,-42.440,179.680,5.686,149.101
C06870=1187.608,-41.494,-42.452,179.683,5.687,149.101
C06871=1187.602,-41.244,-42.464,179.685,5.687,149.100
C06872=1187.597,-40.995,-42.477,179.687,5.687,149.100
C06873=1187.593,-40.745,-42.488,179.690,5.688,149.099
C06874=1187.587,-40.495,-42.500,179.692,5.688,149.098
C06875=1187.582,-40.246,-42.513,179.695,5.689,149.097
C06876=1187.577,-39.996,-42.525,179.696,5.689,149.097
C06877=1187.571,-39.747,-42.537,179.699,5.689,149.096
C06878=1187.566,-39.497,-42.549,179.702,5.689,149.096
C06879=1187.561,-39.247,-42.560,179.704,5.690,149.095
C06880=1187.556,-38.998,-42.573,179.706,5.690,149.094
C06881=1187.551,-38.748,-42.585,179.709,5.690,149.094
C06882=1187.546,-38.499,-42.597,179.711,5.691,149.093
C06883=1187.540,-38.249,-42.609,179.714,5.691,149.092
C06884=1187.535,-37.999,-42.622,179.716,5.692,149.092
C06885=1187.530,-37.750,-42.634,179.718,5.692,149.091
C06886=1187.525,-37.500,-42.646,179.721,5.692,149.090
C06887=1187.520,-37.251,-42.658,179.724,5.693,149.090
C06888=1187.515,-37.000,-42.670,179.726,5.693,149.089
C06889=1187.510,-36.751,-42.683,179.728,5.693,149.089
C06890=1187.505,-36.501,-42.695,179.731,5.694,149.088
C06891=1187.499,-36.251,-42.707,179.733,5.694,149.087
C06892=1187.494,-36.002,-42.720,179.735,5.695,149.087
C06893=1187.489,-35.752,-42.732,179.738,5.695,149.086
C06894=1187.484,-35.503,-42.744,179.740,5.695,149.085
C06895=1187.478,-35.253,-42.756,179.743,5.695,149.085
C06896=1187.473,-35.004,-42.769,179.745,5.696,149.084
C06897=1187.468,-34.754,-42.781,179.748,5.697,149.083
C06898=1187.463,-34.504,-42.793,179.750,5.696,149.083
C06899=1187.457,-34.254,-42.805,179.752,5.697,149.082
C06900=1187.453,-34.004,-42.818,179.755,5.698,149.082
C06901=1187.447,-33.755,-42.831,179.757,5.698,149.081
C06902=1187.442,-33.505,-42.842,179.760,5.698,149.080
C06903=1187.437,-33.256,-42.855,179.762,5.698,149.079
C06904=1187.432,-33.006,-42.867,179.764,5.699,149.079
C06905=1187.426,-32.756,-42.880,179.767,5.699,149.078
C06906=1187.421,-32.507,-42.892,179.769,5.700,149.078
C06907=1187.416,-32.257,-42.904,179.772,5.701,149.077
C06908=1187.411,-32.007,-42.917,179.774,5.700,149.076
C06909=1187.406,-31.758,-42.930,179.776,5.701,149.076
C06910=1187.401,-31.508,-42.941,179.779,5.701,149.075
C06911=1187.396,-31.259,-42.954,179.781,5.702,149.075
C06912=1187.391,-31.009,-42.967,179.784,5.702,149.074
C06913=1187.385,-30.759,-42.979,179.786,5.702,149.073
C06914=1187.381,-30.509,-42.992,179.789,5.703,149.072
C06915=1187.375,-30.260,-43.004,179.791,5.703,149.072
C06916=1187.370,-30.010,-43.016,179.793,5.704,149.071
C06917=1187.365,-29.761,-43.029,179.796,5.704,149.071
C06918=1187.360,-29.511,-43.041,179.798,5.704,149.070
C06919=1187.355,-29.262,-43.054,179.800,5.705,149.069
C06920=1187.350,-29.012,-43.066,179.803,5.705,149.069
C06921=1187.345,-28.762,-43.079,179.806,5.706,149.068
C06922=1187.340,-28.513,-43.091,179.808,5.706,149.067
C06923=1187.334,-28.264,-43.104,179.810,5.706,149.067
C06924=1187.329,-28.014,-43.116,179.813,5.707,149.066
C06925=1187.324,-27.763,-43.129,179.815,5.707,149.065
C06926=1187.319,-27.514,-43.142,179.818,5.708,149.065
C06927=1187.313,-27.265,-43.155,179.820,5.708,149.064
C06928=1187.308,-27.015,-43.166,179.823,5.709,149.064
C06929=1187.303,-26.765,-43.179,179.825,5.709,149.063
C06930=1187.298,-26.515,-43.192,179.827,5.709,149.062
C06931=1187.293,-26.266,-43.205,179.830,5.710,149.062
C06932=1187.288,-26.017,-43.217,179.832,5.710,149.061
C06933=1187.282,-25.767,-43.230,179.835,5.711,149.060
C06934=1187.277,-25.516,-43.243,179.838,5.711,149.060
C06935=1187.272,-25.267,-43.255,179.839,5.711,149.059
C06936=1187.267,-25.018,-43.268,179.842,5.712,149.058
C06937=1187.262,-24.769,-43.280,179.845,5.712,149.058
C06938=1187.258,-24.519,-43.293,179.847,5.713,149.057
C06939=1187.252,-24.269,-43.307,179.849,5.713,149.057
C06940=1187.247,-24.020,-43.319,179.851,5.713,149.056
C06941=1187.242,-23.750,-43.333,179.854,5.714,149.055
C06942=1187.235,-23.481,-43.347,179.857,5.714,149.055
C06943=1187.230,-23.210,-43.360,179.859,5.714,149.054
C06944=1187.225,-22.940,-43.373,179.862,5.715,149.053
C06945=1187.219,-22.691,-43.387,179.865,5.715,149.052
C06946=1187.214,-22.441,-43.399,179.867,5.716,149.052
C06947=1187.209,-22.191,-43.412,179.870,5.717,149.051
C06948=1187.204,-21.942,-43.425,179.872,5.717,149.051
C06949=1187.198,-21.693,-43.438,179.875,5.718,149.050
C06950=1187.193,-21.443,-43.451,179.876,5.718,149.049
C06951=1187.189,-21.193,-43.464,179.879,5.718,149.049
C06952=1187.184,-20.944,-43.476,179.882,5.719,149.048
C06953=1187.178,-20.694,-43.489,179.884,5.719,149.047
C06954=1187.173,-20.444,-43.502,179.887,5.720,149.047
C06955=1187.168,-20.195,-43.515,179.889,5.720,149.046
C06956=1187.163,-19.946,-43.528,179.892,5.721,149.045
C06957=1187.158,-19.695,-43.541,179.894,5.720,149.045
C06958=1187.153,-19.446,-43.554,179.896,5.721,149.044
C06959=1187.148,-19.197,-43.566,179.899,5.722,149.044
C06960=1187.142,-18.946,-43.580,179.902,5.722,149.043
C06961=1187.137,-18.697,-43.592,179.904,5.723,149.042
C06962=1187.132,-18.448,-43.605,179.906,5.723,149.042
C06963=1187.127,-18.197,-43.619,179.909,5.724,149.041
C06964=1187.122,-17.949,-43.632,179.911,5.724,149.040
C06965=1187.117,-17.699,-43.645,179.914,5.724,149.040
C06966=1187.112,-17.449,-43.658,179.916,5.725,149.039
C06967=1187.106,-17.200,-43.671,179.919,5.725,149.038
C06968=1187.101,-16.950,-43.683,179.921,5.726,149.038
C06969=1187.096,-16.700,-43.697,179.924,5.726,149.037
C06970=1187.091,-16.451,-43.709,179.926,5.727,149.037
C06971=1187.086,-16.201,-43.722,179.928,5.727,149.036
C06972=1187.081,-15.952,-43.736,179.931,5.727,149.035
C06973=1187.076,-15.702,-43.749,179.933,5.728,149.035
C06974=1187.071,-15.452,-43.762,179.936,5.729,149.034
C06975=1187.065,-15.203,-43.775,179.938,5.729,149.033
C06976=1187.060,-14.953,-43.788,179.941,5.729,149.033
C06977=1187.055,-14.703,-43.801,179.944,5.730,149.032
C06978=1187.050,-14.454,-43.815,179.946,5.731,149.032
C06979=1187.046,-14.204,-43.828,179.948,5.730,149.031
C06980=1187.040,-13.955,-43.841,179.951,5.731,149.030
C06981=1187.035,-13.705,-43.853,179.953,5.731,149.029
C06982=1187.029,-13.455,-43.867,179.955,5.732,149.029
C06983=1187.025,-13.206,-43.880,179.958,5.733,149.028
C06984=1187.019,-12.956,-43.894,179.961,5.733,149.028
C06985=1187.014,-12.707,-43.906,179.963,5.734,149.027
C06986=1187.010,-12.457,-43.919,179.965,5.734,149.026
C06987=1187.004,-12.208,-43.933,179.968,5.735,149.026
C06988=1186.999,-11.958,-43.946,179.970,5.735,149.025
C06989=1186.994,-11.708,-43.959,179.973,5.735,149.024
C06990=1186.989,-11.459,-43.972,179.975,5.736,149.024
C06991=1186.984,-11.209,-43.986,179.978,5.736,149.023
C06992=1186.979,-10.960,-43.999,179.980,5.737,149.023
C06993=1186.973,-10.709,-44.012,179.983,5.737,149.022
C06994=1186.968,-10.461,-44.026,179.985,5.738,149.021
C06995=1186.963,-10.210,-44.039,179.988,5.739,149.021
C06996=1186.958,-9.961,-44.052,179.991,5.739,149.020
C06997=1186.953,-9.711,-44.066,179.993,5.740,149.020
C06998=1186.948,-9.462,-44.079,179.995,5.740,149.019
C06999=1186.943,-9.212,-44.092,179.997,5.740,149.018
C07000=1186.938,-8.963,-44.106,-180.000,5.740,149.017
C07001=1186.932,-8.713,-44.119,-179.998,5.741,149.017
C07002=1186.928,-8.464,-44.133,-179.995,5.742,149.016
C07003=1186.922,-8.214,-44.146,-179.992,5.742,149.016
C07004=1186.917,-7.964,-44.159,-179.990,5.743,149.015
C07005=1186.912,-7.715,-44.173,-179.988,5.744,149.014
C07006=1186.907,-7.465,-44.186,-179.985,5.744,149.014
C07007=1186.902,-7.216,-44.200,-179.982,5.745,149.013
C07008=1186.897,-6.966,-44.212,-179.980,5.744,149.012
C07009=1186.892,-6.717,-44.227,-179.978,5.745,149.012
C07010=1186.886,-6.467,-44.240,-179.975,5.746,149.011
C07011=1186.882,-6.217,-44.253,-179.973,5.746,149.011
C07012=1186.876,-5.968,-44.267,-179.970,5.746,149.010
C07013=1186.872,-5.718,-44.280,-179.968,5.747,149.009
C07014=1186.866,-5.469,-44.294,-179.965,5.748,149.009
C07015=1186.861,-5.219,-44.307,-179.963,5.748,149.008
C07016=1186.856,-4.970,-44.321,-179.960,5.749,149.007
C07017=1186.851,-4.719,-44.334,-179.958,5.750,149.007
C07018=1186.846,-4.471,-44.347,-179.955,5.750,149.006
C07019=1186.841,-4.220,-44.361,-179.952,5.751,149.005
C07020=1186.835,-3.971,-44.375,-179.950,5.751,149.005
C07021=1186.831,-3.721,-44.388,-179.948,5.751,149.004
C07022=1186.826,-3.472,-44.402,-179.946,5.752,149.004
C07023=1186.820,-3.223,-44.416,-179.943,5.752,149.003
C07024=1186.816,-2.973,-44.429,-179.941,5.753,149.002
C07025=1186.810,-2.724,-44.443,-179.938,5.753,149.002
C07026=1186.805,-2.473,-44.457,-179.935,5.754,149.001
C07027=1186.800,-2.225,-44.470,-179.933,5.754,149.000
C07028=1186.795,-1.974,-44.483,-179.931,5.755,149.000
C07029=1186.790,-1.725,-44.498,-179.928,5.756,148.999
C07030=1186.785,-1.476,-44.511,-179.925,5.756,148.999
C07031=1186.780,-1.226,-44.525,-179.923,5.757,148.998
C07032=1186.774,-0.977,-44.538,-179.921,5.757,148.997
C07033=1186.769,-0.726,-44.552,-179.918,5.758,148.997
C07034=1186.765,-0.477,-44.566,-179.915,5.758,148.996
C07035=1186.759,-0.228,-44.580,-179.913,5.759,148.995
C07036=1186.754,0.022,-44.593,-179.910,5.760,148.995
C07037=1186.750,0.272,-44.607,-179.908,5.760,148.994
C07038=1186.744,0.521,-44.621,-179.906,5.760,148.994
C07039=1186.739,0.771,-44.634,-179.903,5.760,148.993
C07040=1186.733,1.020,-44.648,-179.901,5.761,148.992
C07041=1186.729,1.270,-44.662,-179.898,5.762,148.992
C07042=1186.724,1.519,-44.676,-179.896,5.762,148.991
C07043=1186.718,1.769,-44.689,-179.893,5.763,148.991
C07044=1186.713,2.019,-44.704,-179.891,5.763,148.990
C07045=1186.708,2.288,-44.719,-179.888,5.764,148.989
C07046=1186.703,2.558,-44.734,-179.885,5.764,148.988
C07047=1186.697,2.826,-44.748,-179.882,5.766,148.988
C07048=1186.692,3.095,-44.763,-179.880,5.766,148.987
C07049=1186.687,3.345,-44.777,-179.877,5.767,148.986
C07050=1186.681,3.594,-44.791,-179.875,5.767,148.986
C07051=1186.676,3.844,-44.805,-179.872,5.768,148.985
C07052=1186.671,4.094,-44.819,-179.869,5.768,148.985
C07053=1186.666,4.344,-44.833,-179.867,5.768,148.984
C07054=1186.661,4.592,-44.846,-179.865,5.769,148.983
C07055=1186.656,4.842,-44.861,-179.862,5.769,148.983
C07056=1186.651,5.092,-44.875,-179.860,5.770,148.982
C07057=1186.646,5.341,-44.889,-179.857,5.770,148.981
C07058=1186.641,5.591,-44.902,-179.855,5.771,148.981
C07059=1186.636,5.841,-44.917,-179.852,5.772,148.980
C07060=1186.630,6.090,-44.931,-179.850,5.772,148.980
C07061=1186.626,6.339,-44.944,-179.848,5.773,148.979
C07062=1186.621,6.589,-44.959,-179.845,5.774,148.978
C07063=1186.616,6.839,-44.973,-179.842,5.774,148.978
C07064=1186.610,7.088,-44.987,-179.840,5.775,148.977
C07065=1186.605,7.338,-45.001,-179.837,5.775,148.977
C07066=1186.600,7.588,-45.015,-179.835,5.776,148.976
C07067=1186.595,7.838,-45.029,-179.832,5.776,148.975
C07068=1186.590,8.087,-45.043,-179.829,5.777,148.974
C07069=1186.585,8.336,-45.057,-179.827,5.778,148.974
C07070=1186.580,8.586,-45.071,-179.825,5.778,148.973
C07071=1186.576,8.835,-45.085,-179.822,5.779,148.973
C07072=1186.570,9.084,-45.099,-179.820,5.779,148.972
C07073=1186.565,9.334,-45.113,-179.817,5.780,148.972
C07074=1186.560,9.584,-45.127,-179.815,5.780,148.971
C07075=1186.555,9.834,-45.142,-179.812,5.781,148.970
C07076=1186.550,10.083,-45.156,-179.810,5.782,148.970
C07077=1186.545,10.332,-45.170,-179.807,5.782,148.969
C07078=1186.540,10.582,-45.184,-179.804,5.783,148.968
C07079=1186.535,10.832,-45.198,-179.802,5.784,148.968
C07080=1186.530,11.081,-45.213,-179.800,5.784,148.967
C07081=1186.524,11.330,-45.227,-179.797,5.785,148.966
C07082=1186.519,11.580,-45.241,-179.794,5.785,148.966
C07083=1186.514,11.830,-45.255,-179.792,5.786,148.965
C07084=1186.509,12.080,-45.269,-179.789,5.786,148.965
C07085=1186.504,12.329,-45.284,-179.787,5.787,148.964
C07086=1186.499,12.578,-45.298,-179.785,5.788,148.964
C07087=1186.494,12.828,-45.312,-179.782,5.788,148.963
C07088=1186.489,13.078,-45.326,-179.779,5.789,148.962
C07089=1186.484,13.327,-45.341,-179.777,5.789,148.961
C07090=1186.479,13.576,-45.355,-179.775,5.790,148.961
C07091=1186.474,13.825,-45.369,-179.772,5.791,148.960
C07092=1186.469,14.075,-45.384,-179.769,5.791,148.960
C07093=1186.464,14.325,-45.398,-179.767,5.792,148.959
C07094=1186.458,14.575,-45.413,-179.764,5.792,148.959
C07095=1186.453,14.825,-45.427,-179.762,5.793,148.958
C07096=1186.449,15.074,-45.442,-179.759,5.793,148.957
C07097=1186.444,15.323,-45.456,-179.757,5.794,148.957
C07098=1186.438,15.572,-45.470,-179.754,5.795,148.956
C07099=1186.433,15.822,-45.485,-179.752,5.795,148.955
C07100=1186.428,16.072,-45.499,-179.750,5.796,148.955
C07101=1186.423,16.322,-45.513,-179.746,5.797,148.954
C07102=1186.419,16.571,-45.528,-179.744,5.798,148.954
C07103=1186.414,16.820,-45.542,-179.741,5.798,148.953
C07104=1186.408,17.070,-45.557,-179.739,5.799,148.952
C07105=1186.403,17.320,-45.572,-179.736,5.800,148.952
C07106=1186.398,17.568,-45.586,-179.734,5.800,148.951
C07107=1186.393,17.818,-45.600,-179.731,5.801,148.951
C07108=1186.388,18.068,-45.615,-179.729,5.802,148.950
C07109=1186.383,18.318,-45.629,-179.726,5.802,148.949
C07110=1186.378,18.567,-45.644,-179.723,5.803,148.949
C07111=1186.372,18.817,-45.659,-179.721,5.803,148.948
C07112=1186.368,19.066,-45.673,-179.719,5.804,148.947
C07113=1186.363,19.316,-45.687,-179.716,5.804,148.947
C07114=1186.358,19.565,-45.702,-179.714,5.805,148.946
C07115=1186.353,19.815,-45.717,-179.711,5.806,148.946
C07116=1186.347,20.065,-45.732,-179.709,5.806,148.945
C07117=1186.342,20.313,-45.746,-179.706,5.807,148.944
C07118=1186.337,20.563,-45.760,-179.704,5.808,148.944
C07119=1186.332,20.813,-45.775,-179.701,5.808,148.943
C07120=1186.327,21.062,-45.790,-179.698,5.809,148.942
C07121=1186.322,21.312,-45.805,-179.696,5.809,148.942
C07122=1186.317,21.561,-45.820,-179.694,5.810,148.941
C07123=1186.312,21.811,-45.834,-179.690,5.811,148.941
C07124=1186.307,22.060,-45.848,-179.688,5.812,148.940
C07125=1186.302,22.310,-45.864,-179.686,5.813,148.939
C07126=1186.297,22.560,-45.878,-179.683,5.813,148.939
C07127=1186.292,22.809,-45.893,-179.680,5.814,148.938
C07128=1186.287,23.058,-45.907,-179.678,5.814,148.938
C07129=1186.282,23.308,-45.922,-179.675,5.815,148.937
C07130=1186.277,23.557,-45.937,-179.673,5.815,148.936
C07131=1186.272,23.807,-45.951,-179.671,5.816,148.936
C07132=1186.267,24.057,-45.967,-179.668,5.817,148.935
C07133=1186.262,24.306,-45.981,-179.665,5.817,148.934
C07134=1186.257,24.555,-45.996,-179.663,5.818,148.934
C07135=1186.252,24.805,-46.011,-179.661,5.819,148.933
C07136=1186.247,25.054,-46.026,-179.658,5.819,148.933
C07137=1186.242,25.304,-46.040,-179.655,5.821,148.932
C07138=1186.237,25.553,-46.055,-179.652,5.821,148.932
C07139=1186.231,25.803,-46.070,-179.650,5.822,148.931
C07140=1186.227,26.052,-46.085,-179.647,5.822,148.930
C07141=1186.222,26.302,-46.100,-179.645,5.823,148.930
C07142=1186.216,26.552,-46.115,-179.642,5.824,148.929
C07143=1186.211,26.801,-46.129,-179.640,5.824,148.928
C07144=1186.206,27.051,-46.145,-179.638,5.825,148.928
C07145=1186.201,27.300,-46.160,-179.635,5.826,148.927
C07146=1186.196,27.549,-46.174,-179.632,5.826,148.927
C07147=1186.191,27.799,-46.190,-179.630,5.827,148.926
C07148=1186.186,28.049,-46.204,-179.628,5.827,148.925
C07149=1186.180,28.317,-46.221,-179.624,5.829,148.925
C07150=1186.175,28.586,-46.237,-179.622,5.829,148.924
C07151=1186.170,28.855,-46.253,-179.619,5.830,148.923
C07152=1186.164,29.124,-46.269,-179.616,5.831,148.923
C07153=1186.160,29.373,-46.284,-179.614,5.832,148.922
C07154=1186.155,29.623,-46.300,-179.611,5.832,148.922
C07155=1186.150,29.873,-46.314,-179.608,5.833,148.921
C07156=1186.145,30.122,-46.330,-179.606,5.834,148.920
C07157=1186.140,30.371,-46.345,-179.603,5.834,148.920
C07158=1186.134,30.621,-46.360,-179.601,5.835,148.919
C07159=1186.130,30.870,-46.375,-179.599,5.836,148.919
C07160=1186.124,31.120,-46.390,-179.596,5.836,148.918
C07161=1186.119,31.369,-46.404,-179.593,5.837,148.917
C07162=1186.115,31.618,-46.419,-179.591,5.838,148.917
C07163=1186.109,31.868,-46.435,-179.588,5.839,148.916
C07164=1186.105,32.118,-46.450,-179.585,5.839,148.915
C07165=1186.099,32.368,-46.465,-179.583,5.840,148.915
C07166=1186.095,32.617,-46.480,-179.581,5.841,148.914
C07167=1186.089,32.866,-46.496,-179.578,5.841,148.914
C07168=1186.085,33.115,-46.511,-179.575,5.842,148.913
C07169=1186.079,33.365,-46.526,-179.573,5.843,148.913
C07170=1186.074,33.614,-46.541,-179.570,5.844,148.912
C07171=1186.070,33.864,-46.557,-179.567,5.844,148.911
C07172=1186.064,34.114,-46.572,-179.565,5.845,148.911
C07173=1186.060,34.363,-46.587,-179.562,5.846,148.910
C07174=1186.054,34.613,-46.602,-179.560,5.846,148.909
C07175=1186.049,34.862,-46.617,-179.558,5.847,148.909
C07176=1186.044,35.111,-46.633,-179.555,5.848,148.908
C07177=1186.040,35.361,-46.648,-179.552,5.848,148.908
C07178=1186.034,35.611,-46.664,-179.550,5.850,148.907
C07179=1186.029,35.860,-46.679,-179.547,5.850,148.906
C07180=1186.024,36.109,-46.694,-179.544,5.851,148.906
C07181=1186.019,36.359,-46.709,-179.542,5.852,148.905
C07182=1186.014,36.608,-46.724,-179.540,5.852,148.905
C07183=1186.009,36.858,-46.740,-179.537,5.853,148.904
C07184=1186.004,37.108,-46.756,-179.535,5.854,148.904
C07185=1185.999,37.357,-46.771,-179.532,5.855,148.903
C07186=1185.994,37.606,-46.786,-179.529,5.855,148.902
C07187=1185.989,37.855,-46.801,-179.527,5.856,148.902
C07188=1185.984,38.105,-46.817,-179.524,5.857,148.901
C07189=1185.979,38.355,-46.833,-179.521,5.857,148.900
C07190=1185.974,38.604,-46.848,-179.519,5.858,148.900
C07191=1185.969,38.853,-46.863,-179.517,5.859,148.899
C07192=1185.964,39.103,-46.879,-179.513,5.860,148.899
C07193=1185.960,39.353,-46.894,-179.511,5.861,148.898
C07194=1185.954,39.602,-46.910,-179.509,5.861,148.898
C07195=1185.949,39.851,-46.925,-179.506,5.862,148.897
C07196=1185.945,40.101,-46.941,-179.504,5.863,148.896
C07197=1185.939,40.351,-46.956,-179.501,5.863,148.896
C07198=1185.934,40.600,-46.972,-179.498,5.865,148.895
C07199=1185.929,40.849,-46.988,-179.496,5.866,148.895
C07200=1185.925,41.099,-47.003,-179.493,5.866,148.894
C07201=1185.919,41.349,-47.018,-179.491,5.867,148.893
C07202=1185.914,41.598,-47.034,-179.488,5.867,148.893
C07203=1185.909,41.847,-47.049,-179.486,5.868,148.892
C07204=1185.904,42.097,-47.065,-179.483,5.870,148.892
C07205=1185.899,42.347,-47.081,-179.480,5.870,148.891
C07206=1185.894,42.596,-47.096,-179.478,5.871,148.890
C07207=1185.890,42.845,-47.112,-179.476,5.872,148.890
C07208=1185.884,43.095,-47.128,-179.473,5.872,148.889
C07209=1185.879,43.344,-47.143,-179.470,5.873,148.889
C07210=1185.874,43.593,-47.159,-179.468,5.874,148.888
C07211=1185.870,43.843,-47.174,-179.465,5.875,148.887
C07212=1185.864,44.093,-47.190,-179.462,5.875,148.887
C07213=1185.859,44.342,-47.206,-179.460,5.876,148.886
C07214=1185.854,44.591,-47.222,-179.457,5.877,148.886
C07215=1185.849,44.841,-47.238,-179.454,5.878,148.885
C07216=1185.844,45.090,-47.253,-179.452,5.879,148.885
C07217=1185.840,45.340,-47.269,-179.449,5.879,148.884
C07218=1185.834,45.589,-47.284,-179.447,5.880,148.883
C07219=1185.829,45.838,-47.301,-179.445,5.881,148.883
C07220=1185.824,46.088,-47.317,-179.441,5.882,148.882
C07221=1185.819,46.338,-47.332,-179.439,5.883,148.882
C07222=1185.814,46.587,-47.347,-179.437,5.884,148.881
C07223=1185.810,46.836,-47.364,-179.434,5.884,148.880
C07224=1185.804,47.086,-47.379,-179.432,5.885,148.880
C07225=1185.800,47.336,-47.395,-179.429,5.886,148.879
C07226=1185.794,47.585,-47.411,-179.426,5.887,148.879
C07227=1185.789,47.834,-47.427,-179.424,5.888,148.878
C07228=1185.784,48.084,-47.443,-179.421,5.888,148.877
C07229=1185.779,48.333,-47.459,-179.419,5.889,148.877
C07230=1185.775,48.582,-47.475,-179.416,5.890,148.876
C07231=1185.770,48.832,-47.490,-179.413,5.891,148.876
C07232=1185.764,49.081,-47.506,-179.411,5.892,148.875
C07233=1185.760,49.331,-47.523,-179.408,5.892,148.875
C07234=1185.755,49.580,-47.538,-179.406,5.893,148.874
C07235=1185.749,49.830,-47.554,-179.403,5.895,148.873
C07236=1185.745,50.079,-47.571,-179.400,5.895,148.873
C07237=1185.739,50.329,-47.586,-179.398,5.896,148.872
C07238=1185.735,50.578,-47.603,-179.396,5.896,148.872
C07239=1185.729,50.827,-47.618,-179.392,5.898,148.871
C07240=1185.725,51.078,-47.634,-179.390,5.899,148.871
C07241=1185.720,51.326,-47.651,-179.388,5.899,148.870
C07242=1185.714,51.576,-47.666,-179.385,5.900,148.869
C07243=1185.710,51.825,-47.683,-179.383,5.901,148.869
C07244=1185.704,52.075,-47.699,-179.380,5.902,148.868
C07245=1185.701,52.324,-47.715,-179.377,5.903,148.868
C07246=1185.695,52.573,-47.730,-179.375,5.903,148.867
C07247=1185.690,52.823,-47.746,-179.372,5.904,148.866
C07248=1185.685,53.072,-47.762,-179.369,5.906,148.866
C07249=1185.680,53.323,-47.779,-179.367,5.906,148.865
C07250=1185.675,53.571,-47.795,-179.364,5.907,148.865
C07251=1185.670,53.821,-47.811,-179.362,5.907,148.864
C07252=1185.665,54.070,-47.828,-179.359,5.909,148.863
C07253=1185.659,54.339,-47.845,-179.356,5.909,148.863
C07254=1185.655,54.607,-47.863,-179.354,5.910,148.862
C07255=1185.649,54.876,-47.880,-179.351,5.912,148.862
C07256=1185.644,55.144,-47.897,-179.348,5.912,148.861
C07257=1185.639,55.394,-47.913,-179.345,5.913,148.860
C07258=1185.634,55.643,-47.929,-179.343,5.914,148.860
C07259=1185.629,55.893,-47.946,-179.340,5.915,148.859
C07260=1185.624,56.141,-47.962,-179.338,5.916,148.859
C07261=1185.619,56.391,-47.978,-179.335,5.916,148.858
C07262=1185.614,56.641,-47.995,-179.332,5.918,148.857
C07263=1185.609,56.891,-48.011,-179.330,5.918,148.857
C07264=1185.604,57.139,-48.027,-179.327,5.919,148.856
C07265=1185.599,57.389,-48.044,-179.325,5.921,148.856
C07266=1185.594,57.638,-48.059,-179.322,5.921,148.855
C07267=1185.589,57.888,-48.076,-179.319,5.922,148.855
C07268=1185.585,58.137,-48.093,-179.317,5.923,148.854
C07269=1185.579,58.387,-48.108,-179.314,5.924,148.854
C07270=1185.574,58.637,-48.125,-179.312,5.925,148.853
C07271=1185.569,58.885,-48.142,-179.309,5.925,148.852
C07272=1185.564,59.135,-48.158,-179.307,5.926,148.852
C07273=1185.559,59.384,-48.174,-179.304,5.928,148.851
C07274=1185.555,59.634,-48.191,-179.301,5.928,148.851
C07275=1185.550,59.882,-48.207,-179.299,5.929,148.850
C07276=1185.544,60.133,-48.224,-179.296,5.929,148.850
C07277=1185.540,60.382,-48.240,-179.293,5.931,148.849
C07278=1185.535,60.631,-48.257,-179.291,5.932,148.848
C07279=1185.530,60.881,-48.273,-179.288,5.932,148.848
C07280=1185.525,61.130,-48.289,-179.286,5.934,148.847
C07281=1185.520,61.380,-48.306,-179.283,5.934,148.847
C07282=1185.515,61.629,-48.323,-179.280,5.935,148.846
C07283=1185.510,61.878,-48.339,-179.278,5.936,148.846
C07284=1185.506,62.128,-48.356,-179.275,5.937,148.845
C07285=1185.499,62.377,-48.372,-179.273,5.938,148.844
C07286=1185.495,62.627,-48.389,-179.270,5.939,148.844
C07287=1185.490,62.876,-48.405,-179.268,5.940,148.843
C07288=1185.485,63.125,-48.422,-179.265,5.941,148.843
C07289=1185.480,63.375,-48.439,-179.262,5.941,148.842
C07290=1185.476,63.624,-48.455,-179.260,5.942,148.842
C07291=1185.470,63.874,-48.471,-179.257,5.944,148.841
C07292=1185.466,64.123,-48.488,-179.255,5.945,148.841
C07293=1185.461,64.373,-48.505,-179.252,5.945,148.840
C07294=1185.455,64.622,-48.521,-179.249,5.947,148.839
C07295=1185.451,64.871,-48.538,-179.247,5.947,148.839
C07296=1185.446,65.121,-48.555,-179.244,5.948,148.838
C07297=1185.441,65.370,-48.572,-179.241,5.950,148.838
C07298=1185.436,65.619,-48.588,-179.239,5.950,148.837
C07299=1185.431,65.869,-48.605,-179.237,5.951,148.837
C07300=1185.426,66.118,-48.622,-179.233,5.952,148.836
C07301=1185.421,66.367,-48.638,-179.231,5.953,148.835
C07302=1185.416,66.617,-48.656,-179.229,5.954,148.835
C07303=1185.411,66.866,-48.672,-179.226,5.954,148.834
C07304=1185.407,67.115,-48.689,-179.223,5.956,148.834
C07305=1185.401,67.365,-48.706,-179.221,5.956,148.833
C07306=1185.396,67.614,-48.722,-179.219,5.957,148.833
C07307=1185.391,67.864,-48.740,-179.215,5.959,148.832
C07308=1185.387,68.113,-48.756,-179.213,5.960,148.832
C07309=1185.382,68.363,-48.773,-179.211,5.960,148.831
C07310=1185.376,68.612,-48.790,-179.207,5.961,148.830
C07311=1185.372,68.861,-48.806,-179.205,5.962,148.830
C07312=1185.367,69.111,-48.824,-179.203,5.963,148.829
C07313=1185.362,69.361,-48.840,-179.200,5.965,148.829
C07314=1185.357,69.609,-48.857,-179.197,5.965,148.828
C07315=1185.352,69.859,-48.874,-179.195,5.966,148.828
C07316=1185.347,70.109,-48.891,-179.192,5.967,148.827
C07317=1185.342,70.358,-48.908,-179.190,5.968,148.827
C07318=1185.337,70.607,-48.925,-179.187,5.969,148.826
C07319=1185.332,70.856,-48.942,-179.184,5.970,148.825
C07320=1185.328,71.106,-48.959,-179.182,5.971,148.825
C07321=1185.323,71.356,-48.976,-179.179,5.972,148.824
